(* CODESYS project plc_chalet_vision_fw15.library
   Title: CHALET_Vision
   Version: 3.0.1
   Placeholder: CHALET_Vision
   Company: Beckhoff CH

Project tree, tasks and I/O mapping:
  libraries: CHALET_BaseComponents, * (Beckhoff CH); Tc2_EtherCAT, * (Beckhoff Automation GmbH); Tc2_Standard, * (Beckhoff Automation GmbH); Tc2_System, * (Beckhoff Automation GmbH); Tc2_Utilities, * (Beckhoff Automation GmbH); Tc3_EventLogger, * (Beckhoff Automation GmbH); Tc3_Module, * (Beckhoff Automation GmbH); Tc3_Vision, * (Beckhoff Automation GmbH)
  COMPONENTs/
    CameraTriggerController/
      Base FB/
        function block FB_CameraTriggerController_Base [ST]: FB_init, Feedback, NextPossibleTriggerTime, Operational, Reset, SetParent, State, Trigger
        interface I_CameraTriggerController_Base: Feedback, NextPossibleTriggerTime, Operational, Reset, SetParent, State
        interface I_CameraTriggerController_StatusOnly: Feedback, Operational, State
      EL2258 - 8Ch. digital output timestamp/
        function block FB_EL2258_1Ch_TSO [ST]: Duration_1us, Operational, Reset, State, Trigger, TriggerDelay_1ns, Update
      EL2596 - 1Ch. LED output and camera trigger/
        function block FB_EL2596 [ST]: Duration_1us, Operational, Reset, State, Trigger, TriggerDelay_1ns, Update
        interface I_HwTimestamp_Mode: Duration_1us, Trigger, TriggerDelay_1ns
      EtherCAT Timestamp trigger/
        function block FB_EtherCAT_Trigger [ST]: NextPossibleTriggerTime, Operational, Reset, State, Trigger, TriggerDelay_1ns, Update
        function block FB_EtherCAT_Trigger_old [ST]: Operational, Reset, State, Trigger, TriggerDelay_1ns, Update
        interface I_SwTimestamp_Mode: Trigger, TriggerDelay_1ns
      GigE - Softwaretrigger/
        function block FB_GigeSoftwaretrigger [ST]: Duration_1us, GigeCamera, Reset, Trigger, TriggerDelay_1ns, Update
        interface I_GigeSoftTrigger_Mode: GigeCamera, Trigger, TriggerDelay_1ns
    IlluminationController/
      EL2595 - 1Ch. LED output timestamp/
        function block FB_EL2595 [ST]: Busy, Duration_1us, Operational, Reset, State, Trigger, Update
      SingleOutput/
        function block FB_IlluminationSingleOutput [ST]: Busy, Configure, FB_init, Initialize, Operational, Reset, State, Trigger, Update
        interface I_IlluminationSingleOutput_Mode: Duration_1us, Trigger
      VIx2000/
        DUTs/
          data type E_VIx2000_Status
          data type ST_VIx2000_Channel
          data type ST_VIx2000_InDevice
          data type ST_VIx2000_OutDevice
          data type ST_VIx2000_Pulse
        function block FB_VIx2000 [ST]: Busy, Configure, Duration_1us, Enable, Initialize, Operational, Reset, State, Trigger, Update
        interface I_VIx2000_Mode: Configure, Trigger
      function block FB_IlluminationController_Base [ST]: Busy, NextPossibleTriggerTime, Operational, Reset, SetParent, State, Trigger
      interface I_IlluminationController_Base: Busy, NextPossibleTriggerTime, Operational, Reset, SetParent, State
      interface I_IlluminationController_StatusOnly: Busy, Operational, State
    ImageProvider/
      Base FB/
        function block FB_ImageProvider_Base [ST]: FB_init, Feedback, Initialize, Operational, Reset, SetParent, State, TryGetImage
        interface I_ImageProvider_Base: Feedback, Operational, Reset, SetParent, State, TryGetImage
        interface I_ImageProvider_StatusOnly: Feedback, Operational, State
      Camera/
        data type E_CameraRegisters_Beckhoff
        data type E_DeviceDefaultState
        data type E_TriggerSource
        function block FB_GigE_Beckhoff [ST]: DeviceDefaultState, DeviceModeNamel, DeviceSerialNumber, DeviceVendorName, DeviceVersion, Exposure_1us, IPAddress, MacAddress, TriggerSource, FB_init, GevCameraControl, Initialize, OID, Reset, Softtrigger, State, TryGetImage, Update
        function block FB_GigE_Vision [ST]: Exposure_1us, FB_init, GevCameraControl, Initialize, OID, Reset, Softtrigger, State, TryGetImage, Update
        interface I_GigEVision_Mode: Exposure_1us, Softtrigger
        interface I_GigEVision_Register_Connection: OID
      ImageFromFile/
        function block FB_ImageFromFile [ST]: FileSourceControl, Initialize, LastImageFileName, OID, RequestSpecificImageName, Reset, State, Trigger, TryGetImage, Update
        interface I_ImageFromFile_Mode: RequestSpecificImageName, Trigger
    Mode/
      Combined illumination and camera triggers/
        function block FB_VisionMode_Pulse_combined [ST]: Configure, Initialize, LastTriggerTime, Name, TriggerAtDcTime, TriggerNow
        interface I_VisionMode_Pulse_combined: Configure, LastTriggerTime, NextPossibleTriggerTime, TriggerAtDcTime, TriggerNow
      Separate illumination and camera triggers/
        function block FB_VisionMode_Pulse_separate [ST]: Configure, Initialize, LastTriggerTime_Camera, LastTriggerTime_Illumination, Name, TriggerAtDcTime_Camera, TriggerAtDcTime_Illumination, TriggerNow_Camera, TriggerNow_Illumination
        interface I_VisionMode_Pulse_separate: Configure, LastTriggerTime_Camera, LastTriggerTime_Illumination, NextPossibleTriggerTime, TriggerAtDcTime_Camera, TriggerAtDcTime_Illumination, TriggerNow_Camera, TriggerNow_Illumination
      function block FB_VisionMode_Base [ST]: LinkComponents, Name, NextPossibleTriggerTime
      interface I_VisionMode_Base: LinkComponents, Name
      interface I_VisionMode_StatusOnly: Name
    VisionSystem/
      function block FB_VisionSystem [ST]: ActiveMode, CameraController, IlluminationController1, IlluminationController2, ImageProvider, FB_exit, ActiveModeName, SetMode, Busy, Error, FB_init, Initialize, Initialized, OID, Operational, Reset, TaskCycleTimeNs, TryGetImage, Update
      interface I_VisionSystem: ActiveMode, CameraController, IlluminationController1, IlluminationController2, ImageProvider, SetMode, Busy, Error, Initialized, Operational, Reset, TaskCycleTimeNs, TryGetImage
    VnRegister-Access/
      internal/
        function block FB_VnRegister_Base [ST]: Error, FB_init, Initialize, OID, ReadDone, Update, WriteDone
        interface I_VnRegister_Status: ReadDone, WriteDone
      function block FB_VnRegister_Memory [ST]: FB_init, ReadData, Update, WriteData
      function block FB_VnRegister_REAL [ST]: FB_init, Update, Value
      function block FB_VnRegister_UDINT [ST]: FB_init, Update, Value
      function block FB_VnRegister_ULINT [ST]: FB_init, Update, Value
  FUNCTIONs/
    Casting/
      function ToCameraController [ST]
      function ToGigeSoftTrigger_Mode [ST]
      function ToGigEVision_Mode [ST]
      function ToHwTimestamp_Mode [ST]
      function ToIlluminationSingleOutput_Mode [ST]
      function ToImageFromFile_Mode [ST]
      function ToImageProvider [ST]
      function TolluminationController [ST]
      function ToSwTimestamp_Mode [ST]
      function ToVisionMode_Pulse_combined [ST]
      function ToVisionMode_Pulse_separate [ST]
      function ToVIx2000_Mode [ST]
    Color/
      data type E_Color_ARGB
      function F_ColorEnumToVector4 [ST]
    Sharpness/
      function F_VND_Sharpness_SumModifiedLaplace_ULINT [ST]
  TYPEs/
    data type E_StateTerminal
    data type ST_ImageWithInfo
  00000000-0000-0000-0000-000000000000|LICENSE.md
  LICENSE.md
  global variables VisionParameterlist
*)

// COMPONENTs/IlluminationController/VIx2000/DUTs/E_VIx2000_Status
{attribute 'qualified_only'}
{attribute 'strict'}
{attribute 'to_string'}
TYPE E_VIx2000_Status :
(
	INIT := 0,
	READY,
	TRIGGERING,
	ERROR,
	RESET,
	RESETING
):=INIT;
END_TYPE

// COMPONENTs/IlluminationController/VIx2000/DUTs/ST_VIx2000_Channel
TYPE ST_VIx2000_Channel :
STRUCT
	nBrightness 	 : UINT;
	nDuration_1us 	 : UDINT;
END_STRUCT
END_TYPE

// COMPONENTs/IlluminationController/VIx2000/DUTs/ST_VIx2000_InDevice
TYPE ST_VIx2000_InDevice :
STRUCT
	bReady					: BOOL := FALSE;		// Illumination ready
	bWarning				: BOOL := FALSE;		// Illumination has warning
	bError					: BOOL := FALSE;		// Illumination has error
	bDiag					: BOOL := FALSE;		// ???
	nStatus					: UDINT := 0;			// Illumination state
	nSwitch_on_counter		: UDINT := 0;			// Illumination switching counter
END_STRUCT
END_TYPE

// COMPONENTs/IlluminationController/VIx2000/DUTs/ST_VIx2000_OutDevice
TYPE ST_VIx2000_OutDevice :
STRUCT
	bEnable					: BOOL 	:= FALSE;					// Illumination enable
	bReset					: BOOL	:= FALSE;					// Illumination reset
END_STRUCT
END_TYPE

// COMPONENTs/IlluminationController/VIx2000/DUTs/ST_VIx2000_Pulse
TYPE ST_VIx2000_Pulse :
STRUCT
	nTimestamp 		: T_DCTIME64;
	nFlashDelay 	: UINT;
END_STRUCT
END_TYPE

// COMPONENTs/ImageProvider/Camera/E_CameraRegisters_Beckhoff
{attribute 'qualified_only'}
{attribute 'to_string'}
TYPE E_CameraRegisters_Beckhoff :
(
BootStrap_VersionMajor_BootStrap_VersionMinor := 16#00000000, // GigE Vision Minor Version
BootStrap_DeviceEndianess_BootStrap_CharacterSet := 16#00000004, // BootStrap CharacterSet
BootStrap_MACAddress_High      := 16#00000008, // None
BootStrap_MACAddress_Low       := 16#0000000C, // None
BootStrap_SupportedLLA_BootStrap_SupportedDHCP_BootStrap_SupportedPersistentIP := 16#00000010, // PersistentIP Register
BootStrap_EnabledDHCP_BootStrap_EnabledPersistentIP_BootStrap_EnabledLLA := 16#00000014, // LLA Register Enabled
BootStrap_IPAddress            := 16#00000024, // Current IP Address Register
BootStrap_SubnetMask           := 16#00000034, // Current Subnet Mask Register
BootStrap_Gateway              := 16#00000044, // Current Subnet Mask Register
DeviceVendorName               := 16#00000048, // Name of the camera vendor which is always Beckhoff Automation GmbH & Co.KG
DeviceModelName                := 16#00000068, // Displays the device model name.
DeviceVersion                  := 16#00000088, // Displays the device version which includes the firmware release and build.
DeviceSerialNumber             := 16#000000D8, // Displays the factory set camera serial number.
DeviceUserID                   := 16#000000E8, // A user set ID of up to 15 characters. By default this field is set to the serial number of the camera.
GevFirstURL                    := 16#00000200, // NULL-terminated string providing the first URL to the XML device description file.
GevSecondURL                   := 16#00000400, // NULL-terminated string providing the second URL to the XML device description file.
BootStrap_NumberOfInterfaces   := 16#00000600, // Number Of Interfaces
BootStrap_PersistentIPAddress  := 16#0000064C, // Persistent IP Address Register
BootStrap_PersistentSubnetMask := 16#0000065C, // Persistent Subnet Mask Register
BootStrap_PersistentDefaultGateway := 16#0000066C, // Persistent Default Gateway Register
BootStrap_MessageChannelCount  := 16#00000900, // Number of Message Channel Register
BootStrap_StreamChannelCount   := 16#00000904, // Number of Stream Channel Register
BootStrap_EVENTDATASupported_BootStrap_WRITEMEMSupported_BootStrap_UserDefinedNameSupported_BootStrap_SerialNumberSupported_BootStrap_ConcatenationSupported_BootStrap_PACKETRESENDSupported_BootStrap_EVENTSupported := 16#00000934, // EVENT Supported
BootStrap_GevHeartbeatTimeout  := 16#00000938, // Current heartbeat timeout in milliseconds
BootStrap_TimestampTickFrequencyHigh := 16#0000093C, // 32-MSB of the timestamp Frequency
BootStrap_TimestampTickFrequencyLow := 16#00000940, // 32-LSB of the timestamp Frequencyy
BootStrap_GevTimestampControl  := 16#00000944, // Timestamp Control Register
BootStrap_TimestampValueHigh   := 16#00000948, // 32-MSB of the timestamp Value
BootStrap_TimestampValueLow    := 16#0000094C, // 32-LSB of the timestamp Value
BootStrap_GVSPExtendedID       := 16#00000960, // GVSP Extended ID
pGevSCPSPacketSizeReg          := 16#00000D04, // None
pGevSCPDReg                    := 16#00000D08, // Inter-Packet Delay
pPhysicalWidthReg              := 16#10000008, // None
pPhysicalHeightReg             := 16#1000000C, // None
pSensorPixelWidthReg           := 16#10000010, // None
pSensorPixelHeightReg          := 16#10000014, // None
pDeviceScanTypeReg             := 16#10000018, // None
pSensorShutterModeReg          := 16#1000001C, // None
pMaxThroughputReg              := 16#10000020, // None
pPixelFormatReg                := 16#10000034, // None
pAcquisitionModeReg            := 16#10000040, // None
pAcquisitionFrameCountReg      := 16#10000044, // None
pSensorColorReg                := 16#10000048, // True, if a color sensor has been detected.
pSensorPolarizationReg         := 16#1000004C, // True, if a polarization sensor has been detected.
pAcquisitionStartReg           := 16#100000A8, // None
pAcquisitionStopReg            := 16#100000AC, // None
pAcquisitionAbortReg           := 16#100000B0, // None
SensorName                     := 16#10000150, // Displays the model of the sensor.
pAcquisitionStatusBaseReg      := 16#10000204, // None
pAcquisitionStatusAcquisitionActiveReg := 16#10000208, // None
pRegion0WidthReg               := 16#10000300, // None
pRegion1WidthReg               := 16#10000304, // None
pRegion2WidthReg               := 16#10000308, // None
pRegion3WidthReg               := 16#1000030C, // None
pRegion4WidthReg               := 16#10000310, // None
pRegion5WidthReg               := 16#10000314, // None
pRegion6WidthReg               := 16#10000318, // None
pRegion7WidthReg               := 16#1000031C, // None
pRegion0MinWidthReg            := 16#10000330, // None
pRegion1MinWidthReg            := 16#10000334, // None
pRegion2MinWidthReg            := 16#10000338, // None
pRegion3MinWidthReg            := 16#1000033C, // None
pRegion4MinWidthReg            := 16#10000340, // None
pRegion5MinWidthReg            := 16#10000344, // None
pRegion6MinWidthReg            := 16#10000348, // None
pRegion7MinWidthReg            := 16#1000034C, // None
pRegion0MaxWidthReg            := 16#10000360, // None
pRegion1MaxWidthReg            := 16#10000364, // None
pRegion2MaxWidthReg            := 16#10000368, // None
pRegion3MaxWidthReg            := 16#1000036C, // None
pRegion4MaxWidthReg            := 16#10000370, // None
pRegion5MaxWidthReg            := 16#10000374, // None
pRegion6MaxWidthReg            := 16#10000378, // None
pRegion7MaxWidthReg            := 16#1000037C, // None
pRegion0IncWidthReg            := 16#10000390, // None
pRegion1IncWidthReg            := 16#10000394, // None
pRegion2IncWidthReg            := 16#10000398, // None
pRegion3IncWidthReg            := 16#1000039C, // None
pRegion4IncWidthReg            := 16#10000400, // None
pRegion5IncWidthReg            := 16#10000404, // None
pRegion6IncWidthReg            := 16#10000408, // None
pRegion7IncWidthReg            := 16#1000040C, // None
pRegion0HeightReg              := 16#10000500, // None
pRegion1HeightReg              := 16#10000504, // None
pRegion2HeightReg              := 16#10000508, // None
pRegion3HeightReg              := 16#1000050C, // None
pRegion4HeightReg              := 16#10000510, // None
pRegion5HeightReg              := 16#10000514, // None
pRegion6HeightReg              := 16#10000518, // None
pRegion7HeightReg              := 16#1000051C, // None
pRegion0MinHeightReg           := 16#10000530, // None
pRegion1MinHeightReg           := 16#10000534, // None
pRegion2MinHeightReg           := 16#10000538, // None
pRegion3MinHeightReg           := 16#1000053C, // None
pRegion4MinHeightReg           := 16#10000540, // None
pRegion5MinHeightReg           := 16#10000544, // None
pRegion6MinHeightReg           := 16#10000548, // None
pRegion7MinHeightReg           := 16#1000054C, // None
pRegion0MaxHeightReg           := 16#10000560, // None
pRegion1MaxHeightReg           := 16#10000564, // None
pRegion2MaxHeightReg           := 16#10000568, // None
pRegion3MaxHeightReg           := 16#1000056C, // None
pRegion4MaxHeightReg           := 16#10000570, // None
pRegion5MaxHeightReg           := 16#10000574, // None
pRegion6MaxHeightReg           := 16#10000578, // None
pRegion7MaxHeightReg           := 16#1000057C, // None
pRegion0IncHeightReg           := 16#10000590, // None
pRegion1IncHeightReg           := 16#10000594, // None
pRegion2IncHeightReg           := 16#10000598, // None
pRegion3IncHeightReg           := 16#1000059C, // None
pRegion4IncHeightReg           := 16#10000600, // None
pRegion5IncHeightReg           := 16#10000604, // None
pRegion6IncHeightReg           := 16#10000608, // None
pRegion7IncHeightReg           := 16#1000060C, // None
pRegion0OffsetXReg             := 16#10000800, // None
pRegion1OffsetXReg             := 16#10000804, // None
pRegion2OffsetXReg             := 16#10000808, // None
pRegion3OffsetXReg             := 16#1000080C, // None
pRegion4OffsetXReg             := 16#10000810, // None
pRegion5OffsetXReg             := 16#10000814, // None
pRegion6OffsetXReg             := 16#10000818, // None
pRegion7OffsetXReg             := 16#1000081C, // None
pRegion0MinOffsetXReg          := 16#10000830, // None
pRegion1MinOffsetXReg          := 16#10000834, // None
pRegion2MinOffsetXReg          := 16#10000838, // None
pRegion3MinOffsetXReg          := 16#1000083C, // None
pRegion4MinOffsetXReg          := 16#10000840, // None
pRegion5MinOffsetXReg          := 16#10000844, // None
pRegion6MinOffsetXReg          := 16#10000848, // None
pRegion7MinOffsetXReg          := 16#1000084C, // None
pRegion0MaxOffsetXReg          := 16#10000860, // None
pRegion1MaxOffsetXReg          := 16#10000864, // None
pRegion2MaxOffsetXReg          := 16#10000868, // None
pRegion3MaxOffsetXReg          := 16#1000086C, // None
pRegion4MaxOffsetXReg          := 16#10000870, // None
pRegion5MaxOffsetXReg          := 16#10000874, // None
pRegion6MaxOffsetXReg          := 16#10000878, // None
pRegion7MaxOffsetXReg          := 16#1000087C, // None
pRegion0IncOffsetXReg          := 16#10000890, // None
pRegion1IncOffsetXReg          := 16#10000894, // None
pRegion2IncOffsetXReg          := 16#10000898, // None
pRegion3IncOffsetXReg          := 16#1000089C, // None
pRegion4IncOffsetXReg          := 16#10000900, // None
pRegion5IncOffsetXReg          := 16#10000904, // None
pRegion6IncOffsetXReg          := 16#10000908, // None
pRegion7IncOffsetXReg          := 16#1000090C, // None
pRegion0OffsetYReg             := 16#10000A00, // None
pRegion1OffsetYReg             := 16#10000A04, // None
pRegion2OffsetYReg             := 16#10000A08, // None
pRegion3OffsetYReg             := 16#10000A0C, // None
pRegion4OffsetYReg             := 16#10000A10, // None
pRegion5OffsetYReg             := 16#10000A14, // None
pRegion6OffsetYReg             := 16#10000A18, // None
pRegion7OffsetYReg             := 16#10000A1C, // None
pRegion0MinOffsetYReg          := 16#10000A30, // None
pRegion1MinOffsetYReg          := 16#10000A34, // None
pRegion2MinOffsetYReg          := 16#10000A38, // None
pRegion3MinOffsetYReg          := 16#10000A3C, // None
pRegion4MinOffsetYReg          := 16#10000A40, // None
pRegion5MinOffsetYReg          := 16#10000A44, // None
pRegion6MinOffsetYReg          := 16#10000A48, // None
pRegion7MinOffsetYReg          := 16#10000A4C, // None
pRegion0MaxOffsetYReg          := 16#10000A60, // None
pRegion1MaxOffsetYReg          := 16#10000A64, // None
pRegion2MaxOffsetYReg          := 16#10000A68, // None
pRegion3MaxOffsetYReg          := 16#10000A6C, // None
pRegion4MaxOffsetYReg          := 16#10000A70, // None
pRegion5MaxOffsetYReg          := 16#10000A74, // None
pRegion6MaxOffsetYReg          := 16#10000A78, // None
pRegion7MaxOffsetYReg          := 16#10000A7C, // None
pRegion0IncOffsetYReg          := 16#10000A90, // None
pRegion1IncOffsetYReg          := 16#10000A94, // None
pRegion2IncOffsetYReg          := 16#10000A98, // None
pRegion3IncOffsetYReg          := 16#10000A9C, // None
pRegion4IncOffsetYReg          := 16#10000B00, // None
pRegion5IncOffsetYReg          := 16#10000B04, // None
pRegion6IncOffsetYReg          := 16#10000B08, // None
pRegion7IncOffsetYReg          := 16#10000B0C, // None
DeviceFirmwareVersion          := 16#10010000, // Displays the currently loaded firmware version manufacturer's code.
pSensorHorizontalDriveModeReg  := 16#11000010, // None
pSensorVerticalDriveModeReg    := 16#11000014, // None
pGevSCPDMinReg                 := 16#12000D08, // Minimum Inter-Packet Delay register
pGevSCPDMaxReg                 := 16#12100D08, // Maximum Inter-Packet Delay register
pGevSCPDIncReg                 := 16#12200D08, // Increment Inter-Packet Delay register
pGevIPConfigurationStatusReg   := 16#20000000, // None
pFrameRateReg                  := 16#30000008, // None
pAcquisitionFrameRateEnableReg := 16#30000010, // None
pGainReg                       := 16#30000014, // None
pOffsetReg                     := 16#3000001C, // None
pExposureModeReg               := 16#30000020, // None
pExposureTimeReg               := 16#30000024, // None
ReverseX_Reg                   := 16#3000005C, // None
ReverseY_Reg                   := 16#30000060, // None
pPixelColorFilterReg           := 16#30000064, // None
pBalanceRatioReg               := 16#30000104, // None
pBalanceRatioRedReg            := 16#30000108, // None
pBalanceRatioGreenReg          := 16#3000010C, // None
pBalanceRatioBlueReg           := 16#30000110, // None
pGammaReg                      := 16#30000300, // None
pTestPatternCountReg           := 16#30000404, // None
pTestPatternReg                := 16#30000408, // None
pTestPatternModeReg            := 16#3000040C, // None
pTestPatternParameter1Reg      := 16#30000410, // None
pTestPatternParameter2Reg      := 16#30000414, // None
pTestPatternHorizontalPositionReg := 16#30000418, // None
pTestPatternVerticalPositionReg := 16#3000041C, // None
pTestPatternHorizontalStepSizeReg := 16#30000420, // None
pTestPatternVerticalStepSizeReg := 16#30000424, // None
pTestPatternHorizontalNumReg   := 16#30000428, // None
pTestPatternVerticalNumReg     := 16#3000042C, // None
pTestPatternColorWidthReg      := 16#30000430, // None
pTestPatternBackGroundReg      := 16#30000434, // None
pTestPatternGradientStepReg    := 16#30000438, // None
pTestPatternParameterMaskReg   := 16#30000440, // None
TestPatternDescription         := 16#30001000, // None
UserSetDescription             := 16#30001120, // Description of the selected User Set content.
UserSetDescription1            := 16#30001140, // Description of the selected User Set content.
UserSetDescription2            := 16#30001160, // Description of the selected User Set content.
UserSetDescription3            := 16#30001180, // Description of the selected User Set content.
UserSetDescription4            := 16#300011A0, // Description of the selected User Set content.
pUserSet0LoadReg               := 16#30001200, // None
pUserSet1LoadReg               := 16#30001204, // None
pUserSet2LoadReg               := 16#30001208, // None
pUserSet3LoadReg               := 16#3000120C, // None
pUserSet4LoadReg               := 16#30001210, // None
pUserSet0SaveReg               := 16#30001300, // None
pUserSet1SaveReg               := 16#30001304, // None
pUserSet2SaveReg               := 16#30001308, // None
pUserSet3SaveReg               := 16#3000130C, // None
pUserSet4SaveReg               := 16#30001310, // None
pUserSetDefaultReg             := 16#30001500, // None
pUserSetFeatureEnableReg       := 16#30001510, // None
pRegionsAvailableReg           := 16#30010000, // Maximum regions of interest available.
pSensorROIMinimumHorizontalValueReg := 16#30010100, // The minimum horizontal value register
pSensorROIMinimumVerticalValueReg := 16#30010104, // The minimum vertical value register
pSensorROIMaximumHorizontalValueReg := 16#30010108, // The maximum horizontal value register
pSensorROIMaximumVerticalValueReg := 16#3001010C, // The maximum vertical value register
pRegionModeReg                 := 16#30010800, // Region Mode base register.
pRegion1ModeReg                := 16#30010804, // Region Mode 1 register.
pRegion2ModeReg                := 16#30010808, // Region Mode 2 register.
pRegion3ModeReg                := 16#3001080C, // Region Mode 3 register.
pRegion4ModeReg                := 16#30010810, // Region Mode 4 register.
pRegion5ModeReg                := 16#30010814, // Region Mode 5 register.
pRegion6ModeReg                := 16#30010818, // Region Mode 6 register.
pRegion7ModeReg                := 16#3001081C, // Region Mode 7 register.
pLineModeReg                   := 16#30020040, // None
pLineInverterReg               := 16#30030040, // None
pLineStatus                    := 16#30040040, // None
pTriggerModeBaseReg            := 16#31000100, // None
pSoftwareTriggerAcquisitionStartReg := 16#31000104, // None
pTriggerSourceBaseReg          := 16#31000108, // None
pTriggerActivationAcquisitionStartReg := 16#3100010C, // None
pTriggerDelayAcquisitionStartReg := 16#31000110, // None
pTriggerModeFrameStartReg      := 16#31000400, // None
pSoftwareTriggerFrameStartReg  := 16#31000404, // None
pTriggerSourceFrameStartReg    := 16#31000408, // None
pTriggerActivationFrameStartReg := 16#3100040C, // None
pTriggerDelayFrameStartReg     := 16#31000410, // None
pFrameRateRegMax               := 16#31001020, // None
pExposureTimeMaxReg            := 16#31001024, // None
pFrameRateRegMin               := 16#31001028, // None
pExposureTimeMinReg            := 16#3100102C, // None
pHorizontalBinningReg          := 16#31001030, // None
pVerticalBinningReg            := 16#31001034, // None
pOpticControllerPresentReg     := 16#32000004, // None
pOpticControllerStatusReg      := 16#32000008, // None
pObjectSensorDistanceReg       := 16#32000010, // Object Sensor Distance Register
pDeviceConnectionSpeedReg      := 16#32100010, // None
pDeviceConnectionStatusReg     := 16#32100014, // None
pDeviceResetReg                := 16#32100018, // None
pDeviceIndicatorModeReg        := 16#32110000, // None
pDeviceStateReg                := 16#32110004, // None
pDeviceDefaultStateReg         := 16#32110008, // None
pLightControllerPresentReg     := 16#33000004, // None
pLightConnectionStatusReg      := 16#33000008, // None
pLightController0Channel1TriggerActiveReg := 16#33000110, // Trigger channel 1 active register
pLightController0Channel2TriggerActiveReg := 16#33000114, // Trigger channel 2 active register
pLightController0Channel3TriggerActiveReg := 16#33000118, // Trigger channel 3 active register
pLightController0Channel4TriggerActiveReg := 16#3300011C, // Trigger channel 4 active register
pLightController0Channel1BrightnessReg := 16#33000120, // Brightness register of channel 1
pLightController0Channel2BrightnessReg := 16#33000124, // Brightness register of channel 2
pLightController0Channel3BrightnessReg := 16#33000128, // Brightness register of channel 3
pLightController0Channel4BrightnessReg := 16#3300012C, // Brightness register of channel 4
pLightController0Channel1TriggerModeReg := 16#33000130, // None
pLightController0Channel2TriggerModeReg := 16#33000134, // None
pLightController0Channel3TriggerModeReg := 16#33000138, // None
pLightController0Channel4TriggerModeReg := 16#3300013C, // None
pLightController0Channel1TriggerDurationReg := 16#33000140, // None
pLightController0Channel2TriggerDurationReg := 16#33000144, // None
pLightController0Channel3TriggerDurationReg := 16#33000148, // None
pLightController0Channel4TriggerDurationReg := 16#3300014C, // None
pLightController0Channel1TriggerDelayReg := 16#33000150, // None
pLightController0Channel2TriggerDelayReg := 16#33000154, // None
pLightController0Channel3TriggerDelayReg := 16#33000158, // None
pLightController0Channel4TriggerDelayReg := 16#3300015C, // None
LightController0Channel1Color  := 16#33001000, // The color of the emitted light.
LightController0Channel2Color  := 16#33001014, // The color of the emitted light.
LightController0Channel3Color  := 16#33001028, // The color of the emitted light.
LightController0Channel4Color  := 16#3300103C, // The color of the emitted light.
pLightControllerEnabledReg     := 16#33100000, // None
pLightControllerPowerGoodReg   := 16#33100004, // None
pLUTEnabledReg                 := 16#35000000, // None
pTransferBlockDurationLowReg   := 16#35000100, // None
pTransferBlockDurationHighReg  := 16#35000104, // None
pTLParamsLockedReg             := 16#35000108, // Features locked during acquisition
pPayloadSizeReg                := 16#3500010C, // None
pPacketSizeMinReg              := 16#36000100, // Minimum packet size register
pPacketSizeMaxReg              := 16#36000104, // Maximum packet size register
pPacketSizeIncReg              := 16#36000108, // Increment of packet size register
pCounter0EventSourceReg        := 16#37000100, // Counter0 Event Source Reg
pCounter1EventSourceReg        := 16#37000104, // Counter1 Event Source Reg
pCounter2EventSourceReg        := 16#37000108, // Counter2 Event Source Reg
pCounter3EventSourceReg        := 16#3700010C, // Counter3 Event Source Reg
pCounter4EventSourceReg        := 16#37000110, // Counter4 Event Source Reg
pCounter5EventSourceReg        := 16#37000114, // Counter5 Event Source Reg
pCounter0ResetReg              := 16#37000200, // Counter0 Reset Reg
pCounter1ResetReg              := 16#37000204, // Counter1 Reset Reg
pCounter2ResetReg              := 16#37000208, // Counter2 Reset Reg
pCounter3ResetReg              := 16#3700020C, // Counter3 Reset Reg
pCounter4ResetReg              := 16#37000210, // Counter4 Reset Reg
pCounter5ResetReg              := 16#37000214, // Counter5 Reset Reg
pCounter0ValueReg              := 16#37000300, // Counter0 Value Reg
pCounter1ValueReg              := 16#37000304, // Counter1 Value Reg
pCounter2ValueReg              := 16#37000308, // Counter2 Value Reg
pCounter3ValueReg              := 16#3700030C, // Counter3 Value Reg
pCounter4ValueReg              := 16#37000310, // Counter4 Value Reg
pCounter5ValueReg              := 16#37000314, // Counter5 Value Reg
pDeviceTemperatureBaseReg      := 16#40000004, // None
pDeviceTemperatureCoreReg      := 16#40000008, // None
pDeviceTemperaturePhyReg       := 16#4000000C, // None
pDeviceTemperatureLiquidLensReg := 16#40000010, // None
pTimestampImage                := 16#41000004, // None
pExtendedInternalTimestampControlRegister := 16#41000050, // None
pExtendedEtherCATTimestampControlRegister := 16#41000054, // None
pTimestampRegHigh              := 16#41000100, // None
pDistributedClocksTimestampRegHigh := 16#41000104, // None
pTimestampLatchRegHigh         := 16#41000110, // None
pDistributedClocksTimestampLatchRegHigh := 16#41000114, // None
pTimestampRegLow               := 16#41000200, // None
pDistributedClocksTimestampRegLow := 16#41000204, // None
pTimestampLatchRegLow          := 16#41000210, // None
pDistributedClocksTimestampLatchRegLow := 16#41000214, // None
pEtherCATLinkActiveReg         := 16#50000000, // None
pGevMACAddressHighWordReg := 16#04F91B00, // None
pGevMACAddressLowWordReg := 16#04F91B04 // None
) UDINT;
END_TYPE

// COMPONENTs/ImageProvider/Camera/E_DeviceDefaultState
{attribute 'qualified_only'}
{attribute 'to_string'}
TYPE E_DeviceDefaultState :
(
	AutoDetect		 	:= 0,
	GigE_Vision	 		:= 1,
	EtherCAT_IO			:= 2,
	EtherCAT_Full		:= 3
)UDINT := AutoDetect;
END_TYPE

// COMPONENTs/ImageProvider/Camera/E_TriggerSource
{attribute 'qualified_only'}
{attribute 'to_string'}
TYPE E_TriggerSource :
(
	SoftwareTrigger 	:= 0,
	HardwareInput	 	:= 1,
	EtherCAT			:= 2
)UDINT := SoftwareTrigger;
END_TYPE

// FUNCTIONs/Color/E_Color_ARGB
TYPE E_Color_ARGB : CHALET_BaseComponents.E_Colors_ARGB; END_TYPE

// TYPEs/E_StateTerminal
{attribute 'qualified_only'}
{attribute 'strict'}
{attribute 'to_string'}
TYPE E_StateTerminal :
(
	RESET := 0,
	RESETING,
	INIT := 10,
	READY := 20,
	TRIGGERING := 30,
	ERROR := 100
):=INIT;
END_TYPE

// TYPEs/ST_ImageWithInfo
TYPE ST_ImageWithInfo :
STRUCT
	ipImage			: ITcVnImage;			// Image
	stInfo 			: TcVnImageInfo;		// Image information   
	sCurrentImageFileName : STRING(500);		// Image name.  For a file the file name, for a camera a fictitious name  
	stGvspInfo 		: GVSP_IMAGE_INFO;		// Returns the GVSP (GigE Vision Streaming Protocol) meta information.
END_STRUCT
END_TYPE

// VisionParameterlist
{attribute 'qualified_only'}
VAR_GLOBAL CONSTANT
	(*Maximum GigE-Register read at same time*)
	MAX_VN_REGISTER_READ 			: UDINT := 1;
	
	(*Maximum GigE-Register write at same time*)
	MAX_VN_REGISTER_WRITE 			: UDINT := 1;
	
	(* The state machine for the illuminaton waits in the “Triggering” state until the component has increased the nSwitch_on_counter *)
	ILLUMINATION_WAIT_FOR_TRIGGER_FEEDBACK : BOOL := FALSE;
END_VAR

// COMPONENTs/CameraTriggerController/Base FB/FB_CameraTriggerController_Base
{attribute 'no_explicit_call' := 'Do not call the body - Stick to OOP'}
FUNCTION_BLOCK ABSTRACT FB_CameraTriggerController_Base EXTENDS FB_CH_Object IMPLEMENTS I_CameraTriggerController_Base
VAR
	ipVisionSystem		: I_VisionSystem;			//Interface to "Owner" of this module. Visionsystem
	fbAlarmGeneral 		: FB_TcAlarm;				// Terminal general alarm
	{attribute 'hide'}  						
	fbFeedback 				: FB_CH_Feedback(THIS^.fbSourceInfo);
END_VAR

METHOD FB_init : BOOL
VAR_INPUT
	bInitRetains : BOOL; // if TRUE, the retain variables are initialized (warm start / cold start)
	bInCopyCode : BOOL;  // if TRUE, the instance afterwards gets moved into the copy code (online change)
END_VAR
VAR_INST
	{attribute 'hide'}
	bFBInitCalledOnce : BOOL; //Do the following code once during start up and not during onlinechange
END_VAR
//Do the following code once during start up and not during onlinechange
IF NOT bFBInitCalledOnce THEN 
	
	;

END_IF

bFBInitCalledOnce := TRUE;
END_METHOD

{attribute 'monitoring':='call'}
PROPERTY Feedback : I_CH_Feedback
GET
Feedback := THIS^.fbFeedback;
END_GET
END_PROPERTY

{attribute 'monitoring' := 'call'}
PROPERTY NextPossibleTriggerTime : T_DCTIME64
GET
VAR
	nEtherCatCycles 	: UINT;	
END_VAR
//If attribute 'TcCallAfterOutputUpdate' is set, it takes 1 cycle more to send timestamp to hardware
IF TwinCAT_SystemInfoVarList._TaskInfo[THIS^.TaskIndex].InCallAfterOutputUpdate THEN
	nEtherCatCycles := 3;
ELSE
	nEtherCatCycles := 2;
END_IF


NextPossibleTriggerTime := F_GetCurDcTaskTime64()(*1ns*) + (THIS^.ipVisionSystem.TaskCycleTimeNs(*1ns*) * nEtherCatCycles (*Cycles*)) + 300_000(*300us(determined by testing)*);
END_GET
END_PROPERTY

{attribute 'monitoring' := 'call'}
PROPERTY Operational : BOOL
GET
Operational := TRUE;
END_GET
END_PROPERTY

METHOD ABSTRACT Reset : HRESULT
END_METHOD

METHOD SetParent
VAR_INPUT
	ipVisionSystem  : I_VisionSystem;
END_VAR
THIS^.ipVisionSystem := ipVisionSystem;
END_METHOD

{attribute 'monitoring' := 'call'}
PROPERTY PUBLIC State : E_StateTerminal
GET
State := E_StateTerminal.READY;
END_GET
END_PROPERTY

METHOD ABSTRACT Trigger : HRESULT
VAR_INPUT
	//The data type T_DCTIME64 represents the distributed clock system time (abbreviated as DC time) as a linear 64-bit integer value. 
	//The time is expressed in nanoseconds since 1/1/2000 UTC. The smallest unit is a nanosecond.
	//F_GetCurDcTickTime64()
	nDCTimeStamp	: T_DCTIME64;
END_VAR
END_METHOD

END_FUNCTION_BLOCK

// COMPONENTs/CameraTriggerController/Base FB/I_CameraTriggerController_Base
INTERFACE I_CameraTriggerController_Base EXTENDS I_CH_Object, I_CameraTriggerController_StatusOnly, __SYSTEM.IQueryInterface

{attribute 'monitoring':='call'}
PROPERTY Feedback : I_CH_Feedback
GET
END_GET
END_PROPERTY

{attribute 'monitoring' := 'call'}
PROPERTY NextPossibleTriggerTime : T_DCTIME64
GET
END_GET
END_PROPERTY

{attribute 'monitoring' := 'call'}
PROPERTY Operational : BOOL
GET
END_GET
END_PROPERTY

METHOD Reset : HRESULT
END_METHOD

METHOD SetParent
VAR_INPUT
	ipVisionSystem  : I_VisionSystem;
END_VAR
END_METHOD

{attribute 'monitoring' := 'call'}
PROPERTY PUBLIC State : E_StateTerminal
GET
END_GET
END_PROPERTY

END_INTERFACE

// COMPONENTs/CameraTriggerController/Base FB/I_CameraTriggerController_StatusOnly
INTERFACE I_CameraTriggerController_StatusOnly EXTENDS __SYSTEM.IQueryInterface

{attribute 'monitoring':='call'}
PROPERTY Feedback : I_CH_Feedback
GET
END_GET
END_PROPERTY

{attribute 'monitoring' := 'call'}
PROPERTY Operational : BOOL
GET
END_GET
END_PROPERTY

{attribute 'monitoring' := 'call'}
PROPERTY PUBLIC State : E_StateTerminal
GET
END_GET
END_PROPERTY

END_INTERFACE

// COMPONENTs/VisionSystem/I_VisionSystem
INTERFACE I_VisionSystem EXTENDS I_CH_Object

{attribute 'monitoring' := 'call'}
PROPERTY ActiveMode : I_VisionMode_StatusOnly
GET
END_GET
END_PROPERTY

{attribute 'monitoring' := 'call'}
PROPERTY CameraController : I_CameraTriggerController_StatusOnly
GET
END_GET
END_PROPERTY

{attribute 'monitoring' := 'call'}
PROPERTY IlluminationController1 : I_IlluminationController_StatusOnly
GET
END_GET
END_PROPERTY

{attribute 'monitoring' := 'call'}
PROPERTY IlluminationController2 : I_IlluminationController_StatusOnly
GET
END_GET
END_PROPERTY

{attribute 'monitoring' := 'call'}
PROPERTY ImageProvider : I_ImageProvider_StatusOnly
GET
END_GET
END_PROPERTY

METHOD SetMode : HRESULT
VAR_INPUT
	ipAnyMode : I_VisionMode_Base;
END_VAR
END_METHOD

{attribute 'monitoring' := 'call'}
//Module already has a task - already a trigger active
PROPERTY ABSTRACT Busy : BOOL
GET
END_GET
END_PROPERTY

{attribute 'monitoring' := 'call'}
PROPERTY Error : BOOL  // Module started successfully and entered aquiring mode
GET
END_GET
END_PROPERTY

{attribute 'monitoring':='call'}
PROPERTY Initialized : BOOL
GET
END_GET
END_PROPERTY

{attribute 'monitoring' := 'call'}
PROPERTY PUBLIC Operational : BOOL // Module started successfully and entered aquiring mode
GET
END_GET
END_PROPERTY

METHOD Reset : HRESULT
VAR_INPUT
END_VAR
END_METHOD

{attribute 'monitoring' := 'call'}
PROPERTY TaskCycleTimeNs : UDINT // Set task cycle time in multiples of 100 ns
GET
END_GET
END_PROPERTY

METHOD TryGetImage : HRESULT
VAR_INPUT
	stImageWithInfo : REFERENCE TO ST_ImageWithInfo;
END_VAR
END_METHOD

END_INTERFACE

// COMPONENTs/Mode/I_VisionMode_StatusOnly
INTERFACE I_VisionMode_StatusOnly EXTENDS __SYSTEM.IQueryInterface

{attribute 'monitoring' := 'call'}
// Name or description of this mode
PROPERTY Name : STRING
GET
END_GET
END_PROPERTY

END_INTERFACE

// COMPONENTs/IlluminationController/I_IlluminationController_StatusOnly
INTERFACE I_IlluminationController_StatusOnly EXTENDS  __SYSTEM.IQueryInterface

{attribute 'monitoring' := 'call'}
PROPERTY Busy : BOOL
GET
END_GET
END_PROPERTY

{attribute 'monitoring' := 'call'}
PROPERTY Operational : BOOL
GET
END_GET
END_PROPERTY

{attribute 'monitoring' := 'call'}
PROPERTY PUBLIC State : E_StateTerminal
GET
END_GET
END_PROPERTY

END_INTERFACE

// COMPONENTs/ImageProvider/Base FB/I_ImageProvider_StatusOnly
INTERFACE I_ImageProvider_StatusOnly EXTENDS __SYSTEM.IQueryInterface

{attribute 'monitoring':='call'}
PROPERTY Feedback : I_CH_Feedback
GET
END_GET
END_PROPERTY

{attribute 'monitoring' := 'call'}
PROPERTY PUBLIC Operational : BOOL
// Module started successfully and entered aquiring mode
GET
END_GET
END_PROPERTY

{attribute 'monitoring' := 'call'}
PROPERTY State : ETcVnCameraState
GET
END_GET
END_PROPERTY

END_INTERFACE

// COMPONENTs/Mode/I_VisionMode_Base
INTERFACE I_VisionMode_Base EXTENDS I_CH_Object, I_VisionMode_StatusOnly, __SYSTEM.IQueryInterface

METHOD LinkComponents : HRESULT
VAR_INPUT
	ipVisionSystem				: I_VisionSystem;
	ipCameraTriggerController	: I_CameraTriggerController_Base;
	ipImageProvider 			: I_ImageProvider_Base;	
	ipIlluminationController1 : I_IlluminationController_Base;
	ipIlluminationController2 : I_IlluminationController_Base;
END_VAR
END_METHOD

{attribute 'monitoring' := 'call'}
// Name or description of this mode
PROPERTY Name : STRING
GET
END_GET
END_PROPERTY

END_INTERFACE

// COMPONENTs/ImageProvider/Base FB/I_ImageProvider_Base
INTERFACE I_ImageProvider_Base EXTENDS I_CH_Object, I_ImageProvider_StatusOnly, __SYSTEM.IQueryInterface

{attribute 'monitoring':='call'}
PROPERTY Feedback : I_CH_Feedback
GET
END_GET
END_PROPERTY

{attribute 'monitoring' := 'call'}
PROPERTY PUBLIC Operational : BOOL
// Module started successfully and entered aquiring mode
GET
END_GET
END_PROPERTY

METHOD Reset : HRESULT
END_METHOD

METHOD SetParent
VAR_INPUT
	ipObject : I_CH_Object;
END_VAR
END_METHOD

{attribute 'monitoring' := 'call'}
PROPERTY State : ETcVnCameraState
GET
END_GET
END_PROPERTY

METHOD TryGetImage : HRESULT
VAR_INPUT
	stImageWithInfo	: REFERENCE TO ST_ImageWithInfo;
END_VAR
END_METHOD

END_INTERFACE

// COMPONENTs/IlluminationController/I_IlluminationController_Base
INTERFACE I_IlluminationController_Base EXTENDS I_CH_Object, I_IlluminationController_StatusOnly, __SYSTEM.IQueryInterface

{attribute 'monitoring' := 'call'}
PROPERTY Busy : BOOL
GET
END_GET
END_PROPERTY

{attribute 'monitoring' := 'call'}
PROPERTY NextPossibleTriggerTime : T_DCTIME64
GET
END_GET
END_PROPERTY

{attribute 'monitoring' := 'call'}
PROPERTY Operational : BOOL
GET
END_GET
END_PROPERTY

METHOD Reset : HRESULT
END_METHOD

METHOD SetParent
VAR_INPUT
	ipVisionSystem  : I_VisionSystem;
END_VAR
END_METHOD

{attribute 'monitoring' := 'call'}
PROPERTY PUBLIC State : E_StateTerminal
GET
END_GET
END_PROPERTY

END_INTERFACE

// COMPONENTs/CameraTriggerController/EL2258 - 8Ch. digital output timestamp/FB_EL2258_1Ch_TSO
{attribute 'no_explicit_call' := 'Do not call the body - Stick to OOP'}
FUNCTION_BLOCK FB_EL2258_1Ch_TSO EXTENDS FB_CameraTriggerController_Base IMPLEMENTS I_HwTimestamp_Mode
VAR
	bOutput					AT %Q* 	: BOOL;					// Desired State of Output
	nStartTime 				AT %Q*	: T_DCTIME64;			// Trigger time stamp
	nActivate				AT %Q*	: USINT; 				// 0 -> 3 use new time in terminal
	
	nImpulseLength 			: UDINT := 20000;   	// Impulse length of the lighting period [in 1us]	
	nTriggerDelay 			: UDINT := 0;			// The given trigger time is delayed by this value. E.g. to wait for the maximum lighting value before taking a picture  [in 1ns]
	{attribute 'hide'}
	eState					: E_StateTerminal;				// Current terminal state
	eTriggerSubState		:(SEQ_WirteTime, SEQ_Activate, SEQ_WaitForTriggerDone, SEQ_TriggerOff, SEQ_Deactivate, SEQ_Done); //setting the trigger takes several Ethercat cycles
END_VAR

{attribute 'monitoring' := 'call'}
PROPERTY Duration_1us : UDINT
GET
Duration_1us := THIS^.nImpulseLength;
END_GET
SET
THIS^.nImpulseLength := Duration_1us;
END_SET
END_PROPERTY

{attribute 'monitoring' := 'call'}
PROPERTY Operational : BOOL
GET
Operational := (THIS^.eState = E_StateTerminal.READY) OR (THIS^.eState = E_StateTerminal.TRIGGERING);
END_GET
END_PROPERTY

METHOD PUBLIC Reset : HRESULT
VAR_INPUT
END_VAR
IF THIS^.eState = E_StateTerminal.ERROR THEN
	fbFeedback.ActiveCommand := 'Reset';
	fbFeedback.Busy := TRUE;	
	
	THIS^.eState := E_StateTerminal.RESET;
END_IF
END_METHOD

{attribute 'monitoring' := 'call'}
PROPERTY PUBLIC State : E_StateTerminal
GET
State := THIS^.eState;
END_GET
END_PROPERTY

METHOD PUBLIC Trigger : HRESULT
VAR_INPUT
	//The data type T_DCTIME64 represents the distributed clock system time (abbreviated as DC time) as a linear 64-bit integer value. 
	//The time is expressed in nanoseconds since 1/1/2000 UTC. The smallest unit is a nanosecond.
	//F_GetCurDcTickTime64()
	nDCTimeStamp	: T_DCTIME64;
END_VAR
(* Check if the trigger is minimum 3 EtherCat cycles in future *)
IF nDCTimeStamp < THIS^.NextPossibleTriggerTime  THEN
	Trigger := E_FAIL;
	RETURN;
END_IF

(* Check if not in wrong state *)
IF NOT (THIS^.eState = E_StateTerminal.READY) THEN
	Trigger := E_FAIL;
	RETURN;
END_IF

fbFeedback.ActiveCommand := 'Trigger';
fbFeedback.Busy := TRUE;	


THIS^.nStartTime := nDCTimeStamp + THIS^.nTriggerDelay;
THIS^.bOutput := TRUE;
THIS^.nActivate := 0;

THIS^.eTriggerSubState := SEQ_WirteTime;
THIS^.eState := E_StateTerminal.TRIGGERING;
Trigger := S_OK;
END_METHOD

{attribute 'monitoring' := 'call'}
// The given trigger time is delayed by this value. E.g. to wait for the maximum lighting value before taking a picture  [in 1ns]
PROPERTY TriggerDelay_1ns : UDINT
GET
TriggerDelay_1ns := THIS^.nTriggerDelay;
END_GET
SET
THIS^.nTriggerDelay := TriggerDelay_1ns;
END_SET
END_PROPERTY

METHOD PUBLIC Update : HRESULT
VAR_INST
	fbTimeout : TON;
END_VAR
(* Check for terminal errors *)
//IF THIS^.bError AND NOT (THIS^.eState = E_StateTerminal.RESET) THEN 
//	THIS^.eState := E_StateTerminal.ERROR;
//END_IF

(* Handle terminal state machine *)
CASE THIS^.eState OF
	(* Reset all control variables *)
	E_StateTerminal.RESET:
		THIS^.eState := E_StateTerminal.RESETING;
		
	(* Reset all control variables *)
	E_StateTerminal.RESETING:
		THIS^.eState := E_StateTerminal.INIT;	
		
	(* Enable terminal if ready *)
	E_StateTerminal.INIT:			
		THIS^.eState := E_StateTerminal.READY;

	
	(* Terminal is ready *)
	E_StateTerminal.READY:
		fbFeedback.Done := TRUE;	
		
		THIS^.nStartTime := 0;
		THIS^.bOutput := FALSE;
		THIS^.nActivate := 0;
		
	(* Terminal is triggering *)
	E_StateTerminal.TRIGGERING:
		CASE eTriggerSubState OF
			SEQ_WirteTime:
				//Wirte TimeStamp, Output and Activate=0 in .Trigger()
				//The next commands are allowed only in the next Ethercat cycle
				eTriggerSubState := SEQ_Activate;
				
			SEQ_Activate:
				// Activate new time
				THIS^.nActivate := 3;
				eTriggerSubState := SEQ_WaitForTriggerDone;
				
			SEQ_WaitForTriggerDone:
				// Trigger is done and PulsOffTime is done
				IF (F_GetCurDcTaskTime64() >= (THIS^.nStartTime + (THIS^.nImpulseLength*1000)(*1ns*))) THEN
					THIS^.bOutput := FALSE;
					THIS^.nActivate := 0;
					eTriggerSubState := SEQ_TriggerOff;
				END_IF
				
			SEQ_TriggerOff:	
				THIS^.nActivate := 3;
				eTriggerSubState := SEQ_Deactivate;
				
			SEQ_Deactivate:	
				IF (F_GetCurDcTaskTime64()(*1ns*) > THIS^.nStartTime) THEN
					eTriggerSubState := SEQ_Done;
					//Ready for next Trigger
					THIS^.eState := E_StateTerminal.READY;
				END_IF

				
			SEQ_Done:
			;
		END_CASE
	
	
	(* Error occured *)	
	E_StateTerminal.ERROR:
		fbFeedback.HR := E_FAIL;	
		IF NOT THIS^.fbAlarmGeneral.bRaised THEN
			THIS^.fbAlarmGeneral.Raise(0);	
		END_IF
		
		IF (THIS^.fbAlarmGeneral.eConfirmationState = TcEventConfirmationState.Confirmed) THEN
			THIS^.Reset();			
		END_IF			
END_CASE

(* Timeout if an state is to long active *)
fbTimeout.IN := (THIS^.eState = E_StateTerminal.INIT) OR (THIS^.eState = E_StateTerminal.RESETING) OR (THIS^.eState = E_StateTerminal.TRIGGERING);
fbTimeout.PT := T#5S;
fbTimeout();
IF fbTimeout.Q THEN
	THIS^.eState := E_StateTerminal.ERROR;
END_IF
END_METHOD

END_FUNCTION_BLOCK

// COMPONENTs/CameraTriggerController/EL2596 - 1Ch. LED output and camera trigger/I_HwTimestamp_Mode
INTERFACE I_HwTimestamp_Mode EXTENDS __SYSTEM.IQueryInterface

{attribute 'monitoring' := 'call'}
PROPERTY Duration_1us : UDINT
GET
END_GET
SET
END_SET
END_PROPERTY

METHOD PUBLIC Trigger : HRESULT
VAR_INPUT
	//The data type T_DCTIME64 represents the distributed clock system time (abbreviated as DC time) as a linear 64-bit integer value. 
	//The time is expressed in nanoseconds since 1/1/2000 UTC. The smallest unit is a nanosecond.
	//F_GetCurDcTickTime64()
	nDCTimeStamp	: T_DCTIME64;
END_VAR
END_METHOD

{attribute 'monitoring' := 'call'}
// The given trigger time is delayed by this value. E.g. to wait for the maximum lighting value before taking a picture  [in 1ns]
PROPERTY TriggerDelay_1ns : UDINT
GET
END_GET
SET
END_SET
END_PROPERTY

END_INTERFACE

// COMPONENTs/CameraTriggerController/EL2596 - 1Ch. LED output and camera trigger/FB_EL2596
{attribute 'no_explicit_call' := 'Do not call the body - Stick to OOP'}
FUNCTION_BLOCK FB_EL2596 EXTENDS FB_CameraTriggerController_Base IMPLEMENTS I_HwTimestamp_Mode
VAR
	bEnable					AT %Q* 	: BOOL;					// Terminal enable
	bTriggerImage 			AT %Q* 	: BOOL;					// Trigger for lighting and camera	 
	bReset					AT %Q*	: BOOL;					// Terminal reset
	
	TimeStamp 				AT %Q*	: T_DCTIME64;				// Trigger time stamp
	
	bReadyToActivate		AT %I*	: BOOL := FALSE;		// Terminal ready
	bWarning				AT %I*	: BOOL := FALSE;		// Terminal has warning
	bError					AT %I*	: BOOL := FALSE;		// Terminal has error
	nOperationCounter		AT %I*  : USINT := 0;			// Terminal switching counter
	
		 
	bEnableCameraTrigger 	AT %Q* 	: BOOL := TRUE;			// Enable trigger to be used for the camera
	nImpulseLength 			AT %Q* 	: UDINT := 20000;   	// Impulse length of the lighting period [in 1us]
	nTriggerDelay 			AT %Q* 	: UDINT := 10;			// Delay between lighting and camera trigger [in 100ns]

	{attribute 'hide'}
	eState							: E_StateTerminal;		// Current terminal state
	
	{attribute 'hide'}
	nOperationCounterAtTriggerStart			: USINT;				// Old operation counter as reference

END_VAR

{attribute 'monitoring' := 'call'}
PROPERTY Duration_1us : UDINT
GET
Duration_1us := THIS^.nImpulseLength;
END_GET
SET
THIS^.nImpulseLength := Duration_1us;
END_SET
END_PROPERTY

{attribute 'monitoring' := 'call'}
PROPERTY Operational : BOOL
GET
Operational := (THIS^.eState = E_StateTerminal.READY) OR (THIS^.eState = E_StateTerminal.TRIGGERING);
END_GET
END_PROPERTY

METHOD PUBLIC Reset : HRESULT
VAR_INPUT
END_VAR
IF THIS^.bError OR (THIS^.eState = E_StateTerminal.ERROR) THEN
	fbFeedback.ActiveCommand := 'Reset';
	fbFeedback.Busy := TRUE;	
	
	THIS^.eState := E_StateTerminal.RESET;
END_IF
END_METHOD

{attribute 'monitoring' := 'call'}
PROPERTY PUBLIC State : E_StateTerminal
GET
State := THIS^.eState;
END_GET
END_PROPERTY

METHOD PUBLIC Trigger : HRESULT
VAR_INPUT
	//The data type T_DCTIME64 represents the distributed clock system time (abbreviated as DC time) as a linear 64-bit integer value. 
	//The time is expressed in nanoseconds since 1/1/2000 UTC. The smallest unit is a nanosecond.
	//F_GetCurDcTickTime64()
	nDCTimeStamp	: T_DCTIME64;
END_VAR
(* Check if the trigger is minimum 3 EtherCat cycles in future *)
IF nDCTimeStamp < THIS^.NextPossibleTriggerTime  THEN
	Trigger := E_FAIL;
	RETURN;
END_IF

(* Check if not in wrong state *)
IF NOT (THIS^.eState = E_StateTerminal.READY) THEN
	Trigger := E_FAIL;
	RETURN;
END_IF

fbFeedback.ActiveCommand := 'Trigger';
fbFeedback.Busy := TRUE;	


THIS^.nOperationCounterAtTriggerStart := THIS^.nOperationCounter;
THIS^.TimeStamp := nDCTimeStamp;
THIS^.eState := E_StateTerminal.TRIGGERING;
Trigger := S_OK;
END_METHOD

{attribute 'monitoring' := 'call'}
// The given trigger time is delayed by this value. E.g. to wait for the maximum lighting value before taking a picture  [in 1ns]
PROPERTY TriggerDelay_1ns : UDINT
GET
TriggerDelay_1ns := THIS^.nTriggerDelay*100;
END_GET
SET
THIS^.nTriggerDelay := TriggerDelay_1ns/100;
END_SET
END_PROPERTY

METHOD PUBLIC Update : HRESULT
VAR_INST
	fbTimeOut : TON;
END_VAR
(* Check for terminal errors *)
IF THIS^.bError AND NOT (THIS^.eState = E_StateTerminal.RESET) THEN 
	THIS^.eState := E_StateTerminal.ERROR;
END_IF

(* Handle terminal state machine *)
CASE THIS^.eState OF
	(* Reset all control variables *)
	E_StateTerminal.RESET:
		THIS^.bReset := TRUE;
		THIS^.bEnable := FALSE;
		THIS^.bTriggerImage := FALSE;
		THIS^.eState := E_StateTerminal.RESETING;
		
	(* Reset all control variables *)
	E_StateTerminal.RESETING:
		THIS^.bReset := FALSE;
		THIS^.bEnable := FALSE;
		THIS^.bTriggerImage := FALSE;
		THIS^.eState := E_StateTerminal.INIT;	
		
	(* Enable terminal if ready *)
	E_StateTerminal.INIT:			
		IF THIS^.bReadyToActivate THEN
			THIS^.bReset := FALSE;
			THIS^.bEnable := TRUE;
			THIS^.fbAlarmGeneral.Clear(0, TRUE);
			THIS^.eState := E_StateTerminal.READY;
		END_IF
	
	(* Terminal is ready *)
	E_StateTerminal.READY:
		fbFeedback.Done := TRUE;	
		
	(* Terminal is triggering *)
	E_StateTerminal.TRIGGERING:
		THIS^.bTriggerImage := TRUE;
		IF THIS^.nOperationCounterAtTriggerStart <> THIS^.nOperationCounter THEN
			THIS^.bTriggerImage := FALSE;
			THIS^.eState := E_StateTerminal.READY;
		END_IF
	
	(* Error occured *)	
	E_StateTerminal.ERROR:
		fbFeedback.HR := E_FAIL;
		IF NOT THIS^.fbAlarmGeneral.bRaised THEN
			THIS^.fbAlarmGeneral.Raise(0);	
		END_IF
		
		IF (THIS^.fbAlarmGeneral.eConfirmationState = TcEventConfirmationState.Confirmed) THEN
			THIS^.Reset();			
		END_IF			
END_CASE

(* Timeout if an state is to long active *)
fbTimeOut.IN := (THIS^.eState = E_StateTerminal.INIT) OR (THIS^.eState = E_StateTerminal.RESETING) OR (THIS^.eState = E_StateTerminal.TRIGGERING);
fbTimeOut.PT := T#5S;
fbTimeOut();
IF fbTimeOut.Q THEN
	THIS^.eState := E_StateTerminal.ERROR;
END_IF
END_METHOD

END_FUNCTION_BLOCK

// COMPONENTs/CameraTriggerController/EtherCAT Timestamp trigger/FB_EtherCAT_Trigger
{attribute 'no_explicit_call' := 'Do not call the body - Stick to OOP'}
FUNCTION_BLOCK FB_EtherCAT_Trigger EXTENDS FB_CameraTriggerController_Base IMPLEMENTS I_SwTimestamp_Mode
VAR
	nStartTime 				AT %Q*	: T_DCTIME64;			// Trigger time stamp
	
	{attribute 'hide'}
	nTriggerDelay 			: UDINT := 0;					// The given trigger time is delayed by this value. E.g. to wait for the maximum lighting value before taking a picture  [in 100ns]
	
	{attribute 'hide'}
	eState					: E_StateTerminal;				// Current terminal state
END_VAR

{attribute 'monitoring' := 'call'}
PROPERTY NextPossibleTriggerTime : T_DCTIME64
GET
VAR
	nEtherCatCycles 	: UINT;	
END_VAR
//If attribute 'TcCallAfterOutputUpdate' is set, it takes 1 cycle more to send timestamp to hardware
IF TwinCAT_SystemInfoVarList._TaskInfo[THIS^.TaskIndex].InCallAfterOutputUpdate THEN
	nEtherCatCycles := 3;
ELSE
	nEtherCatCycles := 2;
END_IF


NextPossibleTriggerTime := F_GetCurDcTaskTime64()(*1ns*) + 3_000_000(*zzz 3ms Beta Firmware*) + (THIS^.ipVisionSystem.TaskCycleTimeNs(*1ns*) * nEtherCatCycles (*Cycles*));
END_GET
END_PROPERTY

{attribute 'monitoring' := 'call'}
PROPERTY Operational : BOOL
GET
Operational := (THIS^.eState = E_StateTerminal.READY) OR (THIS^.eState = E_StateTerminal.TRIGGERING);
END_GET
END_PROPERTY

METHOD PUBLIC Reset : HRESULT
VAR_INPUT
END_VAR
IF THIS^.eState = E_StateTerminal.ERROR THEN
	fbFeedback.ActiveCommand := 'Reset';
	fbFeedback.Busy := TRUE;	

	THIS^.eState := E_StateTerminal.RESET;
END_IF
END_METHOD

{attribute 'monitoring' := 'call'}
PROPERTY PUBLIC State : E_StateTerminal
GET
State := THIS^.eState;
END_GET
END_PROPERTY

METHOD PUBLIC Trigger : HRESULT
VAR_INPUT
	//The data type T_DCTIME64 represents the distributed clock system time (abbreviated as DC time) as a linear 64-bit integer value. 
	//The time is expressed in nanoseconds since 1/1/2000 UTC. The smallest unit is a nanosecond.
	//F_GetCurDcTickTime64()
	nDCTimeStamp	: T_DCTIME64;
END_VAR
(* Check if the trigger is minimum 3 EtherCat cycles in future *)
IF (nDCTimeStamp + THIS^.nTriggerDelay) < THIS^.NextPossibleTriggerTime THEN
	Trigger := E_FAIL;
	RETURN;
END_IF

(* Check if not in wrong state *)
IF NOT (THIS^.eState = E_StateTerminal.READY) THEN
	Trigger := E_FAIL;
	RETURN;
END_IF

fbFeedback.ActiveCommand := 'Trigger';
fbFeedback.Busy := TRUE;	


THIS^.nStartTime := nDCTimeStamp + THIS^.nTriggerDelay;


THIS^.eState := E_StateTerminal.TRIGGERING;
Trigger := S_OK;
END_METHOD

{attribute 'monitoring' := 'call'}
// The given trigger time is delayed by this value. E.g. to wait for the maximum lighting value before taking a picture  [in 1ns]
PROPERTY TriggerDelay_1ns : UDINT
GET
TriggerDelay_1ns := THIS^.nTriggerDelay;
END_GET
SET
THIS^.nTriggerDelay := TriggerDelay_1ns;
END_SET
END_PROPERTY

METHOD PUBLIC Update : HRESULT
VAR_INST
	{attribute 'hide'}
	fbTimeout : TON;
END_VAR
(* Handle terminal state machine *)
CASE THIS^.eState OF
	(* Reset all control variables *)
	E_StateTerminal.RESET:
		//THIS^.bReset := TRUE;
		THIS^.eState := E_StateTerminal.RESETING;
		
	(* Reset all control variables *)
	E_StateTerminal.RESETING:
		//THIS^.bReset := FALSE;
		THIS^.eState := E_StateTerminal.INIT;	
		
	(* Enable terminal if ready *)
	E_StateTerminal.INIT:			
		THIS^.eState := E_StateTerminal.READY;

	(* Terminal is ready *)
	E_StateTerminal.READY:
		fbFeedback.Done := TRUE;
		
		
	(* Terminal is triggering *)
	E_StateTerminal.TRIGGERING:
		//WaitForTriggerDone:
		IF (F_GetCurDcTaskTime64()(*1ns*) >= THIS^.nStartTime) THEN
			THIS^.eState := E_StateTerminal.READY;
		 END_IF
			
	
	(* Error occured *)	
	E_StateTerminal.ERROR:
		fbFeedback.HR := E_FAIL;
		IF NOT THIS^.fbAlarmGeneral.bRaised THEN
			THIS^.fbAlarmGeneral.Raise(0);	
		END_IF
		
		IF (THIS^.fbAlarmGeneral.eConfirmationState = TcEventConfirmationState.Confirmed) THEN
			THIS^.Reset();			
		END_IF			
END_CASE

(* Timeout if an actingstate is to long active *)
fbTimeout.IN := (THIS^.eState = E_StateTerminal.INIT) OR (THIS^.eState = E_StateTerminal.RESETING) OR (THIS^.eState = E_StateTerminal.TRIGGERING);
fbTimeout.PT := T#5S;
fbTimeout();
IF fbTimeout.Q THEN
	THIS^.eState := E_StateTerminal.ERROR;
END_IF
END_METHOD

END_FUNCTION_BLOCK

// COMPONENTs/CameraTriggerController/EtherCAT Timestamp trigger/I_SwTimestamp_Mode
INTERFACE I_SwTimestamp_Mode EXTENDS __SYSTEM.IQueryInterface

METHOD PUBLIC Trigger : HRESULT
VAR_INPUT
	//The data type T_DCTIME64 represents the distributed clock system time (abbreviated as DC time) as a linear 64-bit integer value. 
	//The time is expressed in nanoseconds since 1/1/2000 UTC. The smallest unit is a nanosecond.
	//F_GetCurDcTickTime64()
	nDCTimeStamp	: T_DCTIME64;
END_VAR
END_METHOD

{attribute 'monitoring' := 'call'}
// The given trigger time is delayed by this value. E.g. to wait for the maximum lighting value before taking a picture  [in 1ns]
PROPERTY TriggerDelay_1ns : UDINT
GET
END_GET
SET
END_SET
END_PROPERTY

END_INTERFACE

// COMPONENTs/CameraTriggerController/EtherCAT Timestamp trigger/FB_EtherCAT_Trigger_old
{attribute 'no_explicit_call' := 'Do not call the body - Stick to OOP'}
FUNCTION_BLOCK FB_EtherCAT_Trigger_old EXTENDS FB_CameraTriggerController_Base IMPLEMENTS I_SwTimestamp_Mode
VAR
	nStartTime 				AT %Q*	: T_DCTIME64;			// Trigger time stamp
	nActivate				AT %Q*	: USINT; 				// 0 -> 3 use new time in terminal
	
	{attribute 'hide'}
	nTriggerDelay 			: UDINT := 0;					// The given trigger time is delayed by this value. E.g. to wait for the maximum lighting value before taking a picture  [in 100ns]
	
	{attribute 'hide'}
	eState					: E_StateTerminal;				// Current terminal state
END_VAR

{attribute 'monitoring' := 'call'}
PROPERTY Operational : BOOL
GET
Operational := (THIS^.eState = E_StateTerminal.READY) OR (THIS^.eState = E_StateTerminal.TRIGGERING);
END_GET
END_PROPERTY

METHOD PUBLIC Reset : HRESULT
VAR_INPUT
END_VAR
IF THIS^.eState = E_StateTerminal.ERROR THEN
	fbFeedback.ActiveCommand := 'Reset';
	fbFeedback.Busy := TRUE;	

	THIS^.eState := E_StateTerminal.RESET;
END_IF
END_METHOD

{attribute 'monitoring' := 'call'}
PROPERTY PUBLIC State : E_StateTerminal
GET
State := THIS^.eState;
END_GET
END_PROPERTY

METHOD PUBLIC Trigger : HRESULT
VAR_INPUT
	//The data type T_DCTIME64 represents the distributed clock system time (abbreviated as DC time) as a linear 64-bit integer value. 
	//The time is expressed in nanoseconds since 1/1/2000 UTC. The smallest unit is a nanosecond.
	//F_GetCurDcTickTime64()
	nDCTimeStamp	: T_DCTIME64;
END_VAR
(* Check if the trigger is minimum 3 EtherCat cycles in future *)
IF (nDCTimeStamp + THIS^.nTriggerDelay) < THIS^.NextPossibleTriggerTime THEN
	Trigger := E_FAIL;
	RETURN;
END_IF

(* Check if not in wrong state *)
IF NOT (THIS^.eState = E_StateTerminal.READY) THEN
	Trigger := E_FAIL;
	RETURN;
END_IF

fbFeedback.ActiveCommand := 'Trigger';
fbFeedback.Busy := TRUE;	


THIS^.nStartTime := nDCTimeStamp + THIS^.nTriggerDelay;
THIS^.nActivate := 3; (*Activate*)

THIS^.eState := E_StateTerminal.TRIGGERING;
Trigger := S_OK;
END_METHOD

{attribute 'monitoring' := 'call'}
// The given trigger time is delayed by this value. E.g. to wait for the maximum lighting value before taking a picture  [in 1ns]
PROPERTY TriggerDelay_1ns : UDINT
GET
TriggerDelay_1ns := THIS^.nTriggerDelay;
END_GET
SET
THIS^.nTriggerDelay := TriggerDelay_1ns;
END_SET
END_PROPERTY

METHOD PUBLIC Update : HRESULT
VAR_INST
	{attribute 'hide'}
	fbTimeout : TON;
END_VAR
(* Handle terminal state machine *)
CASE THIS^.eState OF
	(* Reset all control variables *)
	E_StateTerminal.RESET:
		//THIS^.bReset := TRUE;
		THIS^.eState := E_StateTerminal.RESETING;
		
	(* Reset all control variables *)
	E_StateTerminal.RESETING:
		//THIS^.bReset := FALSE;
		THIS^.eState := E_StateTerminal.INIT;	
		
	(* Enable terminal if ready *)
	E_StateTerminal.INIT:			
		THIS^.eState := E_StateTerminal.READY;

	(* Terminal is ready *)
	E_StateTerminal.READY:
		fbFeedback.Done := TRUE;
		THIS^.nActivate := 0;
		
		
	(* Terminal is triggering *)
	E_StateTerminal.TRIGGERING:
		//WaitForTriggerDone:
		IF (F_GetCurDcTaskTime64()(*1ns*) >= (THIS^.nStartTime)) THEN
			//Befor leave triggering, stay 1 cycle in Activate=0
			IF THIS^.nActivate = 0 THEN
				THIS^.eState := E_StateTerminal.READY;
			ELSE 
				THIS^.nActivate := 0;(*Deactivate*)
			END_IF

		 END_IF
			
	
	(* Error occured *)	
	E_StateTerminal.ERROR:
		fbFeedback.HR := E_FAIL;
		IF NOT THIS^.fbAlarmGeneral.bRaised THEN
			THIS^.fbAlarmGeneral.Raise(0);	
		END_IF
		
		IF (THIS^.fbAlarmGeneral.eConfirmationState = TcEventConfirmationState.Confirmed) THEN
			THIS^.Reset();			
		END_IF			
END_CASE

(* Timeout if an actingstate is to long active *)
fbTimeout.IN := (THIS^.eState = E_StateTerminal.INIT) OR (THIS^.eState = E_StateTerminal.RESETING) OR (THIS^.eState = E_StateTerminal.TRIGGERING);
fbTimeout.PT := T#5S;
fbTimeout();
IF fbTimeout.Q THEN
	THIS^.eState := E_StateTerminal.ERROR;
END_IF
END_METHOD

END_FUNCTION_BLOCK

// COMPONENTs/CameraTriggerController/GigE - Softwaretrigger/FB_GigeSoftwaretrigger
{attribute 'no_explicit_call' := 'Do not call the body - Stick to OOP'}
FUNCTION_BLOCK FB_GigeSoftwaretrigger EXTENDS FB_CameraTriggerController_Base IMPLEMENTS I_GigeSoftTrigger_Mode
VAR
	{attribute 'hide'}
	eState							: E_StateTerminal;		// Current terminal state
	nTimeNextTrigger : T_DCTIME64;
	nTriggerDelay : UDINT := 10;			// Delay between lighting and camera trigger [in 1ns]
	ipGigeCamera : I_GigEVision_Mode;
	
END_VAR

PROPERTY Duration_1us : UDINT
GET
END_GET
SET
END_SET
END_PROPERTY

PROPERTY GigeCamera : I_GigEVision_Mode
GET
GigeCamera := ipGigeCamera;
END_GET
SET
ipGigeCamera := GigeCamera;
END_SET
END_PROPERTY

METHOD PUBLIC Reset : HRESULT
VAR_INPUT
END_VAR
IF (THIS^.eState = E_StateTerminal.ERROR) THEN
	fbFeedback.ActiveCommand := 'Reset';
	fbFeedback.Busy := TRUE;	

	THIS^.eState := E_StateTerminal.RESET;
END_IF
END_METHOD

METHOD Trigger : HRESULT
VAR_INPUT
	//The data type T_DCTIME64 represents the distributed clock system time (abbreviated as DC time) as a linear 64-bit integer value. 
	//The time is expressed in nanoseconds since 1/1/2000 UTC. The smallest unit is a nanosecond.
	//F_GetCurDcTickTime64()
	nDCTimeStamp	: T_DCTIME64;
END_VAR
THIS^.nTimeNextTrigger := nDCTimeStamp;
THIS^.eState := E_StateTerminal.TRIGGERING;

fbFeedback.ActiveCommand := 'Trigger';
fbFeedback.Busy := TRUE;	



Trigger := S_OK;
END_METHOD

{attribute 'monitoring' := 'call'}
// The given trigger time is delayed by this value. E.g. to wait for the maximum lighting value before taking a picture  [in 1ns]
PROPERTY TriggerDelay_1ns : UDINT
GET
TriggerDelay_1ns := THIS^.nTriggerDelay;
END_GET
SET
THIS^.nTriggerDelay := TriggerDelay_1ns;
END_SET
END_PROPERTY

METHOD PUBLIC Update : HRESULT
VAR_INST

END_VAR
VAR
	
	fbTaskInfo		 : PlcTaskSystemInfo;
END_VAR
IF THIS^.ipGigeCamera = 0 THEN
	THIS^.eState := E_StateTerminal.ERROR;
END_IF


(* Handle terminal state machine *)
CASE THIS^.eState OF
	(* Reset all control variables *)
	E_StateTerminal.RESET:
		THIS^.eState := E_StateTerminal.RESETING;
		
	(* Reset all control variables *)
	E_StateTerminal.RESETING:
		THIS^.eState := E_StateTerminal.INIT;	
		
	(* Enable terminal if ready *)
	E_StateTerminal.INIT:			
		THIS^.eState := E_StateTerminal.READY;
	
	(* Terminal is ready *)
	E_StateTerminal.READY:
		fbFeedback.Done := TRUE;	
		
	(* Terminal is triggering *)
	E_StateTerminal.TRIGGERING:
		IF (F_GetCurDcTaskTime64()  >=   (THIS^.nTimeNextTrigger - TO_ULINT(THIS^.nTriggerDelay))) THEN
			THIS^.ipGigeCamera.Softtrigger();
			THIS^.eState := E_StateTerminal.READY;
		END_IF
	
	(* Error occured *)	
	E_StateTerminal.ERROR:
		fbFeedback.HR := E_FAIL;
		;

END_CASE
END_METHOD

END_FUNCTION_BLOCK

// COMPONENTs/CameraTriggerController/GigE - Softwaretrigger/I_GigeSoftTrigger_Mode
INTERFACE I_GigeSoftTrigger_Mode EXTENDS __SYSTEM.IQueryInterface

PROPERTY GigeCamera : I_GigEVision_Mode
GET
END_GET
SET
END_SET
END_PROPERTY

METHOD Trigger : HRESULT
VAR_INPUT
	//The data type T_DCTIME64 represents the distributed clock system time (abbreviated as DC time) as a linear 64-bit integer value. 
	//The time is expressed in nanoseconds since 1/1/2000 UTC. The smallest unit is a nanosecond.
	//F_GetCurDcTickTime64()
	nDCTimeStamp	: T_DCTIME64;
END_VAR
END_METHOD

{attribute 'monitoring' := 'call'}
PROPERTY TriggerDelay_1ns : UDINT
GET
END_GET
SET
END_SET
END_PROPERTY

END_INTERFACE

// COMPONENTs/ImageProvider/Camera/I_GigEVision_Mode
INTERFACE I_GigEVision_Mode

{attribute 'monitoring' := 'call'}
PROPERTY Exposure_1us : UDINT
GET
END_GET
SET
END_SET
END_PROPERTY

METHOD PUBLIC Softtrigger : HRESULT
END_METHOD

END_INTERFACE

// COMPONENTs/IlluminationController/EL2595 - 1Ch. LED output timestamp/FB_EL2595
{attribute 'no_explicit_call' := 'Do not call the body - Stick to OOP'}
FUNCTION_BLOCK FB_EL2595 EXTENDS FB_IlluminationController_Base IMPLEMENTS I_IlluminationSingleOutput_Mode
VAR
	(*DOX Control*)
	bOutput					AT %Q* 	: BOOL;					// Desired State of Output
	bReset					AT %Q*	: BOOL;					// Terminal reset
	
	(*DC Sync*)
	nStartTime 				AT %Q*	: T_DCTIME64;			// Trigger time stamp
	nActivate				AT %Q*	: USINT; 				// 0 -> 3 use new time in terminal
	
	(*DOX Status*)
	bReadyToActivate		AT %I*	: BOOL := FALSE;		// Terminal ready
	bWarning				AT %I*	: BOOL := FALSE;		// Terminal has warning
	bError					AT %I*	: BOOL := FALSE;		// Terminal has error
	
	(*DC Feedback*)
	nDCFeedback				AT %I*  : USINT := 0;			// Feedback of outputchanel
	

	nImpulseLength 			AT %Q* 	: UDINT := 20000;   	// Impulse length of the lighting period [in 1us]
	nTriggerDelay 			AT %Q* 	: UDINT := 10;			// Delay between lighting and camera trigger [in 100ns]

	{attribute 'hide'}
	eState					: E_StateTerminal;				// Current terminal state
	eTriggerSubState		:(SEQ_WirteTime, SEQ_Activate, SEQ_WaitForFeedback, SEQ_Done); //setting the trigger takes several Ethercat cycles
END_VAR

{attribute 'monitoring' := 'call'}
//Module already has a task - already a trigger active
PROPERTY Busy : BOOL
GET
Busy := (THIS^.eState = E_StateTerminal.TRIGGERING);
END_GET
END_PROPERTY

{attribute 'monitoring' := 'call'}
PROPERTY Duration_1us : UDINT
GET
Duration_1us := THIS^.nImpulseLength;
END_GET
SET
THIS^.nImpulseLength := Duration_1us;
END_SET
END_PROPERTY

{attribute 'monitoring' := 'call'}
PROPERTY Operational : BOOL
GET
Operational := (THIS^.eState = E_StateTerminal.READY) OR (THIS^.eState = E_StateTerminal.TRIGGERING);
END_GET
END_PROPERTY

METHOD PUBLIC Reset : HRESULT
VAR_INPUT
END_VAR
IF NOT THIS^.Operational THEN
	THIS^.eState := E_StateTerminal.RESET;
END_IF
END_METHOD

{attribute 'monitoring' := 'call'}
PROPERTY PUBLIC State : E_StateTerminal
GET
State := THIS^.eState;
END_GET
END_PROPERTY

METHOD PUBLIC Trigger : HRESULT
VAR_INPUT
	//The data type T_DCTIME64 represents the distributed clock system time (abbreviated as DC time) as a linear 64-bit integer value. 
	//The time is expressed in nanoseconds since 1/1/2000 UTC. The smallest unit is a nanosecond.
	//F_GetCurDcTickTime64()
	nDCTimeStamp	: T_DCTIME64;
END_VAR
(* Check if the trigger is minimum 3 EtherCat cycles in future *)
IF nDCTimeStamp < THIS^.NextPossibleTriggerTime  THEN
	Trigger := E_FAIL;
	RETURN;
END_IF

(* Check if not in wrong state *)
IF NOT (THIS^.eState = E_StateTerminal.READY) THEN
	Trigger := E_FAIL;
	RETURN;
END_IF




THIS^.nStartTime := nDCTimeStamp;
THIS^.bOutput := TRUE;
THIS^.nActivate := 0;

THIS^.eTriggerSubState := SEQ_WirteTime;
THIS^.eState := E_StateTerminal.TRIGGERING;
Trigger := S_OK;
END_METHOD

METHOD PUBLIC Update : HRESULT
VAR_INST
	fbTimeout : TON;
END_VAR
(* Check for terminal errors *)
IF THIS^.bError AND NOT (THIS^.eState = E_StateTerminal.RESET) THEN 
	THIS^.eState := E_StateTerminal.ERROR;
END_IF

(* Handle terminal state machine *)
CASE THIS^.eState OF
	(* Reset all control variables *)
	E_StateTerminal.RESET:
		THIS^.bReset := TRUE;
		THIS^.eState := E_StateTerminal.RESETING;
		
	(* Reset all control variables *)
	E_StateTerminal.RESETING:
		THIS^.bReset := FALSE;
		THIS^.eState := E_StateTerminal.INIT;	
		
	(* Enable terminal if ready *)
	E_StateTerminal.INIT:			
		IF THIS^.bReadyToActivate THEN
			THIS^.bReset := FALSE;
			THIS^.fbAlarmGeneral.Clear(0, TRUE);
			THIS^.eState := E_StateTerminal.READY;
		END_IF
	
	(* Terminal is ready *)
	E_StateTerminal.READY:
		THIS^.nStartTime := 0;
		THIS^.bOutput := FALSE;
		THIS^.nActivate := 0;

	(* Terminal is triggering *)
	E_StateTerminal.TRIGGERING:
		CASE eTriggerSubState OF
			SEQ_WirteTime:
				//Wirte TimeStamp, Output and Activate=0 in .Trigger()
				//The next commands are allowed only in the next Ethercat cycle
				eTriggerSubState := SEQ_Activate;
				
			SEQ_Activate:
				// Activate new time
				THIS^.nActivate := 3;
				eTriggerSubState := SEQ_WaitForFeedback;
				
			SEQ_WaitForFeedback:
				// Trigger is done and PulsOffTime is done
				IF ((F_GetCurDcTaskTime64()(*100ns*) > THIS^.nStartTime) AND THIS^.bReadyToActivate) THEN
					THIS^.nActivate := 0;
					eTriggerSubState := SEQ_Done;
					//Ready for next Trigger
					THIS^.eState := E_StateTerminal.READY;
				END_IF

			SEQ_Done:
			;
		END_CASE
	
	
	(* Error occured *)	
	E_StateTerminal.ERROR:
		IF NOT THIS^.fbAlarmGeneral.bRaised THEN
			THIS^.fbAlarmGeneral.Raise(0);	
		END_IF
		
		IF (THIS^.fbAlarmGeneral.eConfirmationState = TcEventConfirmationState.Confirmed) THEN
			THIS^.Reset();			
		END_IF			
END_CASE

(* Timeout if an state is to long active *)
fbTimeout.IN := (THIS^.eState = E_StateTerminal.INIT) OR (THIS^.eState = E_StateTerminal.RESETING) OR (THIS^.eState = E_StateTerminal.TRIGGERING);
fbTimeout.PT := T#5S;
fbTimeout();
IF fbTimeout.Q THEN
	THIS^.eState := E_StateTerminal.ERROR;
END_IF
END_METHOD

END_FUNCTION_BLOCK

// COMPONENTs/IlluminationController/FB_IlluminationController_Base
{attribute 'no_explicit_call' := 'Do not call the body - Stick to OOP'}
FUNCTION_BLOCK ABSTRACT FB_IlluminationController_Base EXTENDS FB_CH_Object IMPLEMENTS I_IlluminationController_Base
VAR
	ipVisionSystem		: I_VisionSystem;			// Interface to "Owner" of this module. Visionsystem
	fbAlarmGeneral 		: FB_TcAlarm;			// Terminal general alarm
END_VAR

{attribute 'monitoring' := 'call'}
//Module already has a task - already a trigger active
PROPERTY ABSTRACT Busy : BOOL
GET
END_GET
END_PROPERTY

{attribute 'monitoring' := 'call'}
PROPERTY NextPossibleTriggerTime : T_DCTIME64
GET
VAR
	nEtherCatCycles 	: UINT;	
END_VAR
//If attribute 'TcCallAfterOutputUpdate' is set, it takes 1 cycle more to send timestamp to hardware
IF TwinCAT_SystemInfoVarList._TaskInfo[THIS^.TaskIndex].InCallAfterOutputUpdate THEN
	nEtherCatCycles := 3;
ELSE
	nEtherCatCycles := 2;
END_IF


NextPossibleTriggerTime := F_GetCurDcTaskTime64()(*1ns*) + (THIS^.ipVisionSystem.TaskCycleTimeNs(*1ns*) * nEtherCatCycles (*Cycles*)) + 300_000(*300us(determined by testing)*);
END_GET
END_PROPERTY

{attribute 'monitoring' := 'call'}
PROPERTY ABSTRACT Operational : BOOL
GET
END_GET
END_PROPERTY

METHOD ABSTRACT Reset : HRESULT
END_METHOD

METHOD SetParent
VAR_INPUT
	ipVisionSystem  : I_VisionSystem;
END_VAR
THIS^.ipVisionSystem := ipVisionSystem;
END_METHOD

{attribute 'monitoring' := 'call'}
PROPERTY ABSTRACT State : E_StateTerminal
GET
END_GET
END_PROPERTY

METHOD ABSTRACT Trigger : HRESULT
VAR_INPUT
	//The data type T_DCTIME64 represents the distributed clock system time (abbreviated as DC time) as a linear 64-bit integer value. 
	//The time is expressed in nanoseconds since 1/1/2000 UTC. The smallest unit is a nanosecond.
	//F_GetCurDcTickTime64()
	nDCTimeStamp	: T_DCTIME64;
END_VAR
END_METHOD

END_FUNCTION_BLOCK

// COMPONENTs/IlluminationController/SingleOutput/I_IlluminationSingleOutput_Mode
INTERFACE I_IlluminationSingleOutput_Mode

{attribute 'monitoring' := 'call'}
PROPERTY Duration_1us : UDINT
GET
END_GET
SET
END_SET
END_PROPERTY

METHOD  Trigger : HRESULT
VAR_INPUT
	//The data type T_DCTIME64 represents the distributed clock system time (abbreviated as DC time) as a linear 64-bit integer value. 
	//The time is expressed in nanoseconds since 1/1/2000 UTC. The smallest unit is a nanosecond.
	//F_GetCurDcTickTime64()
	nDCTimeStamp	: T_DCTIME64;
END_VAR
END_METHOD

END_INTERFACE

// COMPONENTs/IlluminationController/SingleOutput/FB_IlluminationSingleOutput
FUNCTION_BLOCK FB_IlluminationSingleOutput EXTENDS FB_IlluminationController_Base
VAR
	bTrigger 			AT %Q* 	: BOOL;			// Trigger for lighting
	
	nImpulseLength 		: UINT;   				// Impulse length of the lighting period [ms]
	eState				: E_StateTerminal  := E_StateTerminal.READY;		// Current terminal state
	
	fbTriggerOffDelay	: TOF;
END_VAR

{attribute 'monitoring' := 'call'}
//Module already has a task - already a trigger active
PROPERTY Busy : BOOL
GET
Busy := THIS^.eState = E_StateTerminal.TRIGGERING;
END_GET
END_PROPERTY

METHOD Configure : HRESULT
VAR_INPUT

END_VAR
END_METHOD

METHOD FB_init : BOOL
VAR_INPUT
	bInitRetains : BOOL; // if TRUE, the retain variables are initialized (warm start / cold start)
	bInCopyCode : BOOL;  // if TRUE, the instance afterwards gets moved into the copy code (online change)
	
	nImpulseLength 	: UINT;   	// Impulse length of the lighting period [ms]
END_VAR
VAR_INST
	{attribute 'hide'}
	bFBInitCalledOnce : BOOL; //Do the following code once during start up and not during onlinechange
END_VAR
//Do the following code once during start up and not during onlinechange
IF NOT bFBInitCalledOnce THEN 
	

	THIS^.nImpulseLength 	:= nImpulseLength; 	 	


END_IF

bFBInitCalledOnce := TRUE;
END_METHOD

METHOD Initialize : HRESULT
VAR
	hr : HRESULT;
END_VAR
hr := SUPER^.Initialize();

THIS^.eState := E_StateTerminal.READY;
THIS^.fbTriggerOffDelay.PT := UINT_TO_TIME(THIS^.nImpulseLength);

Initialize := hr;
END_METHOD

{attribute 'monitoring' := 'call'}
PROPERTY Operational : BOOL
GET
Operational := (THIS^.eState = E_StateTerminal.READY) OR (THIS^.eState = E_StateTerminal.TRIGGERING);
END_GET
END_PROPERTY

METHOD  Reset : HRESULT
Reset := S_OK;
END_METHOD

{attribute 'monitoring' := 'call'}
PROPERTY PUBLIC State : E_StateTerminal
GET

State := THIS^.eState;
END_GET
END_PROPERTY

METHOD  Trigger : HRESULT
VAR_INPUT
	//The data type T_DCTIME64 represents the distributed clock system time (abbreviated as DC time) as a linear 64-bit integer value. 
	//The time is expressed in nanoseconds since 1/1/2000 UTC. The smallest unit is a nanosecond.
	//F_GetCurDcTickTime64()
	nDCTimeStamp	: T_DCTIME64;
END_VAR
(* Check if the trigger is minimum 3 EtherCat cycles in future *)
IF nDCTimeStamp < THIS^.NextPossibleTriggerTime  THEN
	Trigger := E_FAIL;
	RETURN;
END_IF

(* The trigger methode can be called in each state. 
Is the output is already set, the off-timer is resetet *)

THIS^.fbTriggerOffDelay.IN := TRUE;;
Trigger := S_OK;
END_METHOD

METHOD PUBLIC Update : HRESULT
(* The trigger methode call be called in each state. 
Is the output is already set, the off-timer is resetet *)

(* Handle terminal state machine *)
CASE THIS^.eState OF
	(* Terminal is ready *)
	E_StateTerminal.READY:
		;		
	(* Terminal is triggering *)
	E_StateTerminal.TRIGGERING:
		;
END_CASE

THIS^.fbTriggerOffDelay();
THIS^.fbTriggerOffDelay.IN := FALSE;

//Set Output
THIS^.bTrigger := THIS^.fbTriggerOffDelay.Q;

//Set State
IF THIS^.bTrigger THEN
	THIS^.eState := E_StateTerminal.TRIGGERING;
ELSE	
	THIS^.eState := E_StateTerminal.READY;
END_IF
END_METHOD

END_FUNCTION_BLOCK

// COMPONENTs/IlluminationController/VIx2000/FB_VIx2000
{attribute 'no_explicit_call' := 'Do not call the body - Stick to OOP'}
FUNCTION_BLOCK FB_VIx2000 EXTENDS FB_IlluminationController_Base IMPLEMENTS I_IlluminationController_Base, I_VIx2000_Mode
VAR
	DeviceInputs 	 		AT %I* 	: ST_VIx2000_InDevice;
	DeviceOutputs			AT %Q*	: ST_VIx2000_OutDevice;		
	Pulse_DC_Outputs		AT %Q*	: ST_VIx2000_Pulse;		
	ChannelOrange 			AT %Q*	: ST_VIx2000_Channel;
	ChannelGreen 			AT %Q*	: ST_VIx2000_Channel;
	ChannelBlue 			AT %Q*	: ST_VIx2000_Channel;
	ChannelInfrared 		AT %Q*	: ST_VIx2000_Channel;
	
	
	{attribute 'hide'}
	bInitDone 						: BOOL;
	{attribute 'hide'}	
	eState							: E_VIx2000_Status;
	{attribute 'hide'}	
	nDuration_1us					: UDINT := 100_000; //Puls duration
	{attribute 'hide'}
	nSwitchOnCounterOnTrigger		: UDINT;				// Old operation counter as reference
	{attribute 'hide'}
	fbFeedBackTrigger 				: FB_CH_Feedback(THIS^.fbSourceInfo);
END_VAR
VAR CONSTANT
	N_MAX_BRIGHTNESS : UINT := 511;
END_VAR

{attribute 'monitoring' := 'call'}
//Module already has a task - already a trigger active
PROPERTY Busy : BOOL
GET
Busy := (THIS^.eState = E_VIx2000_Status.TRIGGERING);
END_GET
END_PROPERTY

METHOD Configure : HRESULT
VAR_INPUT
	nOrange 	: UINT(0..N_MAX_BRIGHTNESS);
	nGreen 		: UINT(0..N_MAX_BRIGHTNESS);
	nBlue 		: UINT(0..N_MAX_BRIGHTNESS);
	nInfrared 	: UINT(0..N_MAX_BRIGHTNESS);
	nDuration_1us : UDINT; //Duration of pulse
END_VAR
THIS^.ChannelOrange.nBrightness := LIMIT(0, nOrange, N_MAX_BRIGHTNESS);
THIS^.ChannelGreen.nBrightness := LIMIT(0, nGreen, N_MAX_BRIGHTNESS);
THIS^.ChannelBlue.nBrightness := LIMIT(0, nBlue, N_MAX_BRIGHTNESS);
THIS^.ChannelInfrared.nBrightness := LIMIT(0, nInfrared, N_MAX_BRIGHTNESS);

THIS^.ChannelOrange.nDuration_1us := nDuration_1us;
THIS^.ChannelGreen.nDuration_1us := nDuration_1us;
THIS^.ChannelBlue.nDuration_1us := nDuration_1us;
THIS^.ChannelInfrared.nDuration_1us := nDuration_1us;

THIS^.nDuration_1us := nDuration_1us;
END_METHOD

{attribute 'monitoring' := 'call'}
PROPERTY Duration_1us : UDINT
GET
Duration_1us := THIS^.nDuration_1us;
END_GET
SET
THIS^.nDuration_1us := Duration_1us;

THIS^.ChannelOrange.nDuration_1us := Duration_1us;
THIS^.ChannelGreen.nDuration_1us := Duration_1us;
THIS^.ChannelBlue.nDuration_1us := Duration_1us;
THIS^.ChannelInfrared.nDuration_1us := Duration_1us;
END_SET
END_PROPERTY

{attribute 'monitoring' := 'call'}
PROPERTY Enable : BOOL
GET
Enable := THIS^.DeviceOutputs.bEnable;
END_GET
END_PROPERTY

METHOD Initialize : HRESULT
VAR
	ipChObject 			: I_CH_OBJECT;
	hr: HRESULT;
END_VAR
hr := SUPER^.Initialize();

//Init some default data 
Configure(
	nOrange:= 50, 
	nGreen:= 50, 
	nBlue:= 50, 
	nInfrared:= 50, 
	nDuration_1us:= 10_000);

IF CheckOk(hr) THEN
	THIS^.bInitDone := TRUE;
END_IF

Initialize := hr;
END_METHOD

{attribute 'monitoring' := 'call'}
PROPERTY Operational : BOOL
GET
Operational := (THIS^.eState = E_VIx2000_Status.READY) OR (THIS^.eState = E_VIx2000_Status.TRIGGERING);
END_GET
END_PROPERTY

METHOD PUBLIC Reset : HRESULT
VAR_INPUT
END_VAR
IF NOT THIS^.Operational THEN
	 THIS^.eState := E_VIx2000_Status.RESET;
END_IF
END_METHOD

{attribute 'monitoring' := 'call'}
PROPERTY PUBLIC State : E_StateTerminal
GET
CASE THIS^.eState OF
	E_VIx2000_Status.INIT:
		State := E_StateTerminal.INIT;
		
	E_VIx2000_Status.READY:
		State := E_StateTerminal.READY;
		
	E_VIx2000_Status.TRIGGERING:
		State := E_StateTerminal.TRIGGERING;
		
	E_VIx2000_Status.ERROR:
		State := E_StateTerminal.ERROR;
		
	E_VIx2000_Status.RESET:
		State := E_StateTerminal.RESET;
		
	E_VIx2000_Status.RESETING:	
		State := E_StateTerminal.RESETING;
END_CASE
END_GET
END_PROPERTY

METHOD Trigger : HRESULT
VAR_INPUT
	//The data type T_DCTIME64 represents the distributed clock system time (abbreviated as DC time) as a linear 64-bit integer value. 
	//The time is expressed in nanoseconds since 1/1/2000 UTC. The smallest unit is a nanosecond.
	//F_GetCurDcTickTime64()
	nDCTimeStamp : T_DCTIME64;
END_VAR
(* Check if the trigger is minimum 3 EtherCat cycles in future *)
IF nDCTimeStamp < THIS^.NextPossibleTriggerTime THEN
	Trigger := E_FAIL;
	RETURN;
END_IF



IF (THIS^.eState = E_VIx2000_Status.READY) THEN
	THIS^.nSwitchOnCounterOnTrigger := THIS^.DeviceInputs.nSwitch_on_counter;
	THIS^.Pulse_DC_Outputs.nTimestamp 	:= nDCTimeStamp;
	THIS^.Pulse_DC_Outputs.nFlashDelay 	:= 0;

	THIS^.eState := E_VIx2000_Status.TRIGGERING;
	
	THIS^.fbFeedbackTrigger.hr := S_OK;
ELSE
	THIS^.fbFeedbackTrigger.hr := E_FAIL;
END_IF

Trigger := THIS^.fbFeedbackTrigger.hr;
END_METHOD

METHOD Update : HRESULT
VAR
	bNewCounterValue : BOOL;
END_VAR
VAR_INST
	{attribute 'hide'}
	nSwitchOnCounterShouldValue : UDINT;
	{attribute 'hide'}
	nSwitchOnCounterLastCycle : UDINT;
	{attribute 'hide'}
	fbTimeOutNoReactionToTrigger : TON;
	{attribute 'hide'}
	fbStateTimeout : TON;
	{attribute 'hide'}
	fbTimeoutAlarm : FB_TcAlarm;
	{attribute 'hide'}
	fbAlarmNoReactionToTrigger : FB_TcAlarm;
	{attribute 'hide'}
	eStateOld : E_VIx2000_Status;
END_VAR
(* Check for terminal errors *)
IF THIS^.DeviceInputs.bError AND NOT ((THIS^.eState = E_VIx2000_Status.RESET) OR (THIS^.eState = E_VIx2000_Status.RESETING))THEN 
	THIS^.eState := E_VIx2000_Status.ERROR;
END_IF

(* Handle terminal state machine *)
CASE THIS^.eState OF
	(* Reset all control variables *)
	E_VIx2000_Status.RESET:
		THIS^.DeviceOutputs.bEnable := FALSE;
		THIS^.DeviceOutputs.bReset := FALSE;
		THIS^.Pulse_DC_Outputs.nTimestamp := 0;		
		THIS^.Pulse_DC_Outputs.nTimestamp := 0;	
		fbTimeoutAlarm.Clear(0,0);	
		fbAlarmNoReactionToTrigger.Clear(0,0);
		THIS^.fbFeedbackTrigger.HR := S_OK;
		
		THIS^.eState := E_VIx2000_Status.RESETING;
		
	(* Reset all control variables *)
	E_VIx2000_Status.RESETING:
		THIS^.DeviceOutputs.bEnable := FALSE;
		THIS^.DeviceOutputs.bReset := TRUE;
		THIS^.eState := E_VIx2000_Status.INIT;
	
	(* Enable terminal if ready *)
	E_VIx2000_Status.INIT:			
		THIS^.DeviceOutputs.bEnable := TRUE;
		THIS^.DeviceOutputs.bReset := FALSE;
		IF THIS^.DeviceInputs.bReady THEN
			THIS^.fbAlarmGeneral.Clear(0, TRUE);
			nSwitchOnCounterShouldValue := THIS^.DeviceInputs.nSwitch_on_counter;
			THIS^.eState := E_VIx2000_Status.READY;
		END_IF
	
	(* Terminal is ready *)
	E_VIx2000_Status.READY:
		;
		
	(* Terminal is triggering *)
	E_VIx2000_Status.TRIGGERING:
	IF VisionParameterlist.ILLUMINATION_WAIT_FOR_TRIGGER_FEEDBACK THEN
		//Wait - timeout if no change
		IF (THIS^.nSwitchOnCounterOnTrigger +1) = THIS^.DeviceInputs.nSwitch_on_counter THEN
			THIS^.eState := E_VIx2000_Status.READY;
		END_IF
	ELSE
		//Do not wait
		IF (F_GetCurDcTaskTime64()  >=  THIS^.Pulse_DC_Outputs.nTimestamp)  THEN
			nSwitchOnCounterShouldValue := nSwitchOnCounterShouldValue + 1;
			THIS^.eState := E_VIx2000_Status.READY;
		END_IF
	END_IF

	
	(* Error occured *)	
	E_VIx2000_Status.ERROR:
		IF NOT THIS^.fbAlarmGeneral.bRaised THEN
			THIS^.fbAlarmGeneral.Raise(0);	
		END_IF
		
		IF (THIS^.fbAlarmGeneral.eConfirmationState = TcEventConfirmationState.Confirmed) THEN
			THIS^.Reset();			
		END_IF			
END_CASE

(* Timeout if an state is to long active *)
fbStateTimeout.IN := (THIS^.eState = eStateOld) AND (THIS^.eState = E_VIx2000_Status.INIT) OR (THIS^.eState = E_VIx2000_Status.RESETING) OR (THIS^.eState = E_VIx2000_Status.TRIGGERING);
eStateOld := THIS^.eState;
fbStateTimeout.PT := T#5S;
fbStateTimeout();
IF fbStateTimeout.Q THEN
	//Raise TC3-Eventlogger Alarm
	IF NOT fbTimeOutAlarm.bRaised THEN
		fbTimeoutAlarm.CreateEx(stEventEntry := TC_EVENTS.CHALET_Vision_Events.TimeOut, bWithConfirmation := FALSE, ipSourceInfo := THIS^.fbSourceInfo);
		fbTimeoutAlarm.ipArguments.AddStringByValue(TO_STRING(THIS^.eState));
		fbTimeoutAlarm.Raise(0);
	END_IF
	
	//Change in alarm state
	THIS^.eState := E_VIx2000_Status.ERROR;
END_IF


//Check that the lighting reacts to the trigger signal within the given time and increments its switch-on counter
IF NOT VisionParameterlist.ILLUMINATION_WAIT_FOR_TRIGGER_FEEDBACK THEN
	bNewCounterValue := nSwitchOnCounterLastCycle <> THIS^.DeviceInputs.nSwitch_on_counter;
	nSwitchOnCounterLastCycle := THIS^.DeviceInputs.nSwitch_on_counter;
	fbTimeOutNoReactionToTrigger.IN := NOT bNewCounterValue AND (nSwitchOnCounterShouldValue <> THIS^.DeviceInputs.nSwitch_on_counter);
	fbTimeOutNoReactionToTrigger.PT := T#5S;
	fbTimeOutNoReactionToTrigger();
	IF fbTimeOutNoReactionToTrigger.Q THEN
		//Raise TC3-Eventlogger Alarm
		IF NOT fbAlarmNoReactionToTrigger.bRaised THEN
			fbAlarmNoReactionToTrigger.CreateEx(stEventEntry := TC_EVENTS.CHALET_Vision_Events.NoReactionToTheTrigger, bWithConfirmation := FALSE, ipSourceInfo := THIS^.fbSourceInfo);
			fbAlarmNoReactionToTrigger.Raise(0);
			nSwitchOnCounterShouldValue := THIS^.DeviceInputs.nSwitch_on_counter;
		END_IF
		
		//Change in alarm state
		THIS^.eState := E_VIx2000_Status.ERROR;
	END_IF
END_IF
END_METHOD

END_FUNCTION_BLOCK

// COMPONENTs/IlluminationController/VIx2000/I_VIx2000_Mode
INTERFACE I_VIx2000_Mode

METHOD Configure : HRESULT
VAR_INPUT
	nOrange 	: UINT(0..511);
	nGreen 		: UINT(0..511);
	nBlue 		: UINT(0..511);
	nInfrared 	: UINT(0..511);
	nDuration_1us : UDINT;
END_VAR
END_METHOD

METHOD Trigger : HRESULT
VAR_INPUT
	//The data type T_DCTIME64 represents the distributed clock system time (abbreviated as DC time) as a linear 64-bit integer value. 
	//The time is expressed in nanoseconds since 1/1/2000 UTC. The smallest unit is a nanosecond.
	//F_GetCurDcTickTime64()
	nDCTimeStamp	: T_DCTIME64;
END_VAR
END_METHOD

END_INTERFACE

// COMPONENTs/ImageProvider/Base FB/FB_ImageProvider_Base
{attribute 'no_explicit_call' := 'Do not call the body - Stick to OOP'}
FUNCTION_BLOCK ABSTRACT FB_ImageProvider_Base EXTENDS FB_CH_Object IMPLEMENTS I_ImageProvider_Base
VAR      	
	{attribute 'hide'}							
    fbCrititcalSection : FB_IecCriticalSection;    						// Internal lock for test & set function                                  	
	{attribute 'hide'}														    		
	eState 				: ETcVnCameraState;		
	{attribute 'hide'}  						
	fbFeedback 			: FB_CH_Feedback(THIS^.fbSourceInfo); 
	{attribute 'hide'}
	fbAlarmOIDNotSet 	: FB_TcAlarm;									// Alarm due to source state	
	{attribute 'hide'}
	ipVisionSystem		: I_CH_Object;									// Interface to "Owner" of this module. Visionsystem
END_VAR

METHOD FB_init : BOOL
VAR_INPUT
	bInitRetains : BOOL; // if TRUE, the retain variables are initialized (warm start / cold start)
	bInCopyCode : BOOL;  // if TRUE, the instance afterwards gets moved into the copy code (online change)
END_VAR
VAR_INST
	{attribute 'hide'}
	bFBInitCalledOnce : BOOL; //Do the following code once during start up and not during onlinechange
END_VAR
//Do the following code once during start up and not during onlinechange
IF NOT bFBInitCalledOnce THEN 
	
	;

END_IF

bFBInitCalledOnce := TRUE;
END_METHOD

{attribute 'monitoring':='call'}
PROPERTY Feedback : I_CH_Feedback
GET
Feedback := THIS^.fbFeedback;
END_GET
END_PROPERTY

METHOD Initialize : HRESULT
Initialize := S_OK;
END_METHOD

{attribute 'monitoring' := 'call'}
PROPERTY PUBLIC Operational : BOOL
// Module started successfully and entered aquiring mode
GET
Operational := (eState = TCVN_CS_ACQUIRING) OR (eState = TCVN_CS_TRIGGERING);
END_GET
END_PROPERTY

METHOD ABSTRACT Reset : HRESULT
END_METHOD

METHOD SetParent
VAR_INPUT
	ipObject : I_CH_Object;
END_VAR
THIS^.ipVisionSystem := ipObject;
END_METHOD

{attribute 'monitoring' := 'call'}
PROPERTY ABSTRACT State : ETcVnCameraState
GET
END_GET
END_PROPERTY

METHOD ABSTRACT TryGetImage : HRESULT
VAR_INPUT
	stImageWithInfo : REFERENCE TO ST_ImageWithInfo;
END_VAR
END_METHOD

END_FUNCTION_BLOCK

// COMPONENTs/ImageProvider/Camera/FB_GigE_Beckhoff
{attribute 'no_explicit_call' := 'Do not call the body - Stick to OOP'}
FUNCTION_BLOCK FB_GigE_Beckhoff EXTENDS FB_ImageProvider_Base IMPLEMENTS I_GigEVision_Mode, I_GigEVision_Register_Connection
VAR
	// This FB provides the basic functionality to control a GigE Vision camera and access its calibration data.
	fbCamera 						: FB_VN_GevCameraControl;	

	{attribute 'hide'}
	bResetCommand	: BOOL;
END_VAR


VAR	
	//GigE-Camera-Register
	//Read/Write
	{attribute 'hide'}
	fbRegAcquisitionMode 		: FB_VnRegister_UDINT(ipCameraConnection := THIS^, nAddress := E_CameraRegisters_Beckhoff.pAcquisitionModeReg, nEndian := 0);
	{attribute 'hide'}
	fbRegTriggerMode	 		: FB_VnRegister_UDINT(ipCameraConnection := THIS^, nAddress := E_CameraRegisters_Beckhoff.pTriggerModeFrameStartReg, nEndian := 0);
	{attribute 'hide'}
	fbRegTriggerSource	 		: FB_VnRegister_UDINT(ipCameraConnection := THIS^, nAddress := E_CameraRegisters_Beckhoff.pTriggerSourceFrameStartReg, nEndian := 0);
	{attribute 'hide'}
	fbRegExposureTime	 		: FB_VnRegister_UDINT(ipCameraConnection := THIS^, nAddress := E_CameraRegisters_Beckhoff.pExposureTimeReg, nEndian := 0);
	{attribute 'hide'}
	fbRegDeviceDefaultState		: FB_VnRegister_UDINT(ipCameraConnection := THIS^, nAddress := E_CameraRegisters_Beckhoff.pDeviceDefaultStateReg, nEndian := 0);
	
	//Read only
	{attribute 'hide'}
	fbRegDeviceVendorName		: FB_VnRegister_Memory(ipCameraConnection := THIS^, nAddress := E_CameraRegisters_Beckhoff.DeviceVendorName, nLength := 32); //String	
	{attribute 'hide'}
	fbRegDeviceModelName	 	: FB_VnRegister_Memory(ipCameraConnection := THIS^, nAddress := E_CameraRegisters_Beckhoff.DeviceModelName, nLength := 32); //String	
	{attribute 'hide'}
	fbRegDeviceVersion	 		: FB_VnRegister_Memory(ipCameraConnection := THIS^, nAddress := E_CameraRegisters_Beckhoff.DeviceVersion, nLength := 32); //String	
	{attribute 'hide'}
	fbRegDeviceSerialNumber	 	: FB_VnRegister_Memory(ipCameraConnection := THIS^, nAddress := E_CameraRegisters_Beckhoff.DeviceSerialNumber, nLength := 16); //String	
	{attribute 'hide'}
	fbRegCurrentIPAddress	 	: FB_VnRegister_UDINT(ipCameraConnection := THIS^, nAddress := E_CameraRegisters_Beckhoff.BootStrap_IPAddress, nEndian := 0);  //T_IPv4AddrArr
	{attribute 'hide'}
	fbRegGevMACAddressHighWord	: FB_VnRegister_UDINT(ipCameraConnection := THIS^, nAddress := E_CameraRegisters_Beckhoff.pGevMACAddressHighWordReg, nEndian := 0);
	{attribute 'hide'}
	fbRegGevMACAddressLowWord	: FB_VnRegister_UDINT(ipCameraConnection := THIS^, nAddress := E_CameraRegisters_Beckhoff.pGevMACAddressLowWordReg, nEndian := 0);

	//List
	{attribute 'hide'}
	fbVnRegisterList 			: FB_CH_List;
END_VAR

{attribute 'monitoring' := 'call'}
PROPERTY DeviceDefaultState : E_DeviceDefaultState
GET
DeviceDefaultState := THIS^.fbRegDeviceDefaultState.Value;
END_GET
SET
IF THIS^.fbRegDeviceDefaultState.Value <> DeviceDefaultState THEN
 	//Set Camera from AQUIRING in OPENED - only on new value
	THIS^.fbCamera.StopAcquisition();
END_IF

THIS^.fbRegDeviceDefaultState.Value := DeviceDefaultState;
END_SET
END_PROPERTY

{attribute 'monitoring' := 'call'}
PROPERTY DeviceModeNamel : STRING
GET
fbRegDeviceModelName.ReadData(ADR(DeviceModeNamel));
END_GET
END_PROPERTY

{attribute 'monitoring' := 'call'}
PROPERTY DeviceSerialNumber : STRING
GET
fbRegDeviceSerialNumber.ReadData(ADR(DeviceSerialNumber));
END_GET
END_PROPERTY

{attribute 'monitoring' := 'call'}
PROPERTY DeviceVendorName : STRING
GET
fbRegDeviceVendorName.ReadData(ADR(DeviceVendorName));
END_GET
END_PROPERTY

{attribute 'monitoring' := 'call'}
PROPERTY DeviceVersion : STRING
GET
fbRegDeviceVersion.ReadData(ADR(DeviceVersion));
END_GET
END_PROPERTY

{attribute 'monitoring' := 'call'}
PROPERTY Exposure_1us : UDINT
GET
Exposure_1us := THIS^.fbRegExposureTime.Value;
END_GET
SET
IF THIS^.fbRegExposureTime.Value <> Exposure_1us THEN
 	//Set Camera from AQUIRING in OPENED - only on new value
	THIS^.fbCamera.StopAcquisition();
END_IF

THIS^.fbRegExposureTime.Value := Exposure_1us;
END_SET
END_PROPERTY

{attribute 'monitoring' := 'call'}
//IP-Adress as STRING(15)
PROPERTY IPAddress : T_IPv4Addr
GET
VAR
	nValueTemp : UDINT;
	stAdressByteArray   : T_IPv4AddrArr; // Byte-Array
END_VAR

IF SIZEOF(fbRegCurrentIPAddress.Value) <> (4*SIZEOF(BYTE)) THEN
	//Error wrond Datatype, Return 0.0.0.0
	IPAddress := F_CreateIPv4Addr(stAdressByteArray);
	RETURN;
END_IF



//store in a temp variable
nValueTemp := fbRegCurrentIPAddress.Value;


//convert to struct(Array of byte)
Tc2_System.MEMCPY(srcAddr:= ADR(nValueTemp)+3, destAddr:= ADR(stAdressByteArray)+0, n:= SIZEOF(BYTE));
Tc2_System.MEMCPY(srcAddr:= ADR(nValueTemp)+2, destAddr:= ADR(stAdressByteArray)+1, n:= SIZEOF(BYTE));
Tc2_System.MEMCPY(srcAddr:= ADR(nValueTemp)+1, destAddr:= ADR(stAdressByteArray)+2, n:= SIZEOF(BYTE));
Tc2_System.MEMCPY(srcAddr:= ADR(nValueTemp)+0, destAddr:= ADR(stAdressByteArray)+3, n:= SIZEOF(BYTE));


IPAddress := F_CreateIPv4Addr(stAdressByteArray); //Byte-Array to String
END_GET
END_PROPERTY

{attribute 'monitoring' := 'call'}
//MAC-Adress from camera
PROPERTY MacAddress : STRING(12)
GET
IF NOT(fbRegGevMACAddressHighWord.ReadDone AND fbRegGevMACAddressLowWord.ReadDone) THEN
	//Wait for first read
	RETURN;
END_IF

MacAddress := Tc2_Standard.CONCAT(
								//This function converts a decimal number into a hexadecimal string (base 16).
								STR1:= Tc2_Utilities.DWORD_TO_HEXSTR(in:= fbRegGevMACAddressHighWord.Value, iPrecision:= 4, bLoCase:= TRUE ), 
								STR2:= Tc2_Utilities.DWORD_TO_HEXSTR(in:= fbRegGevMACAddressLowWord.Value, iPrecision:= 8, bLoCase:= TRUE )
								);
END_GET
END_PROPERTY

{attribute 'monitoring' := 'call'}
PROPERTY TriggerSource : E_TriggerSource
GET
TriggerSource := THIS^.fbRegTriggerSource.Value;
END_GET
SET
IF THIS^.fbRegTriggerSource.Value <> TriggerSource THEN
 	//Set Camera from AQUIRING in OPENED - only on new value
	THIS^.fbCamera.StopAcquisition();
END_IF

fbRegTriggerSource.Value := TriggerSource;
END_SET
END_PROPERTY

METHOD FB_init : BOOL
VAR_INPUT
	bInitRetains : BOOL; // if TRUE, the retain variables are initialized (warm start / cold start)
	bInCopyCode : BOOL;  // if TRUE, the instance afterwards gets moved into the copy code (online change)
END_VAR
VAR_INST
	{attribute 'hide'}
	bFBInitCalledOnce : BOOL; //Do the following code once during start up and not during onlinechange
END_VAR
//Do the following code once during start up and not during onlinechange
IF NOT bFBInitCalledOnce THEN 
	//Read/Write
	fbVnRegisterList.AddObject(fbRegAcquisitionMode);
	fbVnRegisterList.AddObject(fbRegTriggerMode);
	fbVnRegisterList.AddObject(fbRegTriggerSource);
	fbVnRegisterList.AddObject(fbRegExposureTime);
	fbVnRegisterList.AddObject(fbRegDeviceDefaultState);
	
	//Read only
	fbVnRegisterList.AddObject(fbRegDeviceVendorName);
	fbVnRegisterList.AddObject(fbRegDeviceModelName);
	fbVnRegisterList.AddObject(fbRegDeviceVersion);
	fbVnRegisterList.AddObject(fbRegDeviceSerialNumber);
	fbVnRegisterList.AddObject(fbRegCurrentIPAddress);
	fbVnRegisterList.AddObject(fbRegGevMACAddressHighWord);
	fbVnRegisterList.AddObject(fbRegGevMACAddressLowWord);
	

	
	//Prepare for EtherCat-TimeStamp-Trigger use
	fbRegAcquisitionMode.Value 	:=  16#00; 	//Continous
	fbRegTriggerMode.Value		:=  16#01; 	//ON	 
	fbRegTriggerSource.Value	:=  E_TriggerSource.EtherCAT; 	//EtherCat	 
	fbRegDeviceDefaultState.Value	:=  E_DeviceDefaultState.AutoDetect; 
	fbRegExposureTime.Value	 	:= 	15; 	//[us] smallest allowed value
	
	
END_IF

bFBInitCalledOnce := TRUE;
END_METHOD

//Reference to base function block
PROPERTY GevCameraControl : REFERENCE TO FB_VN_GevCameraControl
GET
GevCameraControl REF= THIS^.fbCamera;
END_GET
END_PROPERTY

METHOD Initialize : HRESULT
VAR 
	fbTaskInfo		 : PlcTaskSystemInfo;
END_VAR
VAR_INST
	//This error cannot be reset. Requires a reset cold
	{attribute 'hide'}	
	fbInitError : FB_TcAlarm;
END_VAR
SUPER^.Initialize();


// Object id of ImagePoovider is not set
IF THIS^.fbCamera.oidITcVnGevImageProvider = 0 THEN
	IF NOT fbInitError.bRaised THEN 
		//This error cannot be reset. Requires a reset cold
		fbInitError.CreateEx(stEventEntry:=TC_EVENTS.CHALET_Vision_Events.ObjectIdNotSet, ipSourceInfo := THIS^.fbSourceInfo, bWithConfirmation := FALSE);
		fbInitError.Raise(0);
	END_IF
	Initialize := E_FAIL;
	RETURN;
END_IF
END_METHOD

{attribute 'monitoring' := 'call'}
PROPERTY OID : CHALET_BaseComponents.OTCID
GET
OID := THIS^.fbCamera.oidITcVnGevImageProvider;
END_GET
END_PROPERTY

METHOD Reset : HRESULT
VAR_INPUT
END_VAR
bResetCommand := TRUE;
END_METHOD

METHOD PUBLIC Softtrigger : HRESULT
(* Check if not in wrong state *)
IF NOT ((THIS^.eState = ETcVnCameraState.TCVN_CS_ACQUIRING) OR (THIS^.eState = ETcVnCameraState.TCVN_CS_OPENED)) THEN
	Softtrigger := E_FAIL;
	RETURN;
END_IF


THIS^.eState := ETcVnCameraState.TCVN_CS_TRIGGERING;

// Trigger image
Softtrigger := fbCamera.TriggerImage();
END_METHOD

{attribute 'monitoring' := 'call'}
PROPERTY State : ETcVnCameraState
GET
State := THIS^.eState;
END_GET
END_PROPERTY

METHOD  TryGetImage : HRESULT
VAR_INPUT
	stImageWithInfo : REFERENCE TO ST_ImageWithInfo;
END_VAR
IF NOT __ISVALIDREF(stImageWithInfo) THEN
	//Error, invalide input
	TryGetImage := E_FAIL;
	RETURN;
END_IF


(* Release the old image before overwriting it with the new one *)	
IF stImageWithInfo.ipImage <> 0 THEN
	FW_SafeRelease(ADR(stImageWithInfo.ipImage));
END_IF

(*  Lock the image to prevent multiple access *)
(*	🔒 LOCKED FROM HERE --------------------------------------------- *)
IF THIS^.fbCrititcalSection.Enter() THEN
	
	(* Get current image from camera *)
	TryGetImage := fbCamera.GetCurrentImageWithGvspInfo(
						ipImage := stImageWithInfo.ipImage,
						stGvspInfo := stImageWithInfo.stGvspInfo
						);

	(* Get image info from received image *)
	F_VN_GetImageInfo(	ipImage:=stImageWithInfo.ipImage, 
						stImageInfo:=stImageWithInfo.stInfo, 
						hrPrev:=TryGetImage );
	
	(* for a camera a fictitious name *)
	stImageWithInfo.sCurrentImageFileName := TO_STRING(stImageWithInfo.stGvspInfo.BlockId);			

	(*	🔓 LOCKED TO HERE ----------------------------------------------- *)
	THIS^.fbCrititcalSection.Leave();
END_IF
END_METHOD

METHOD Update : HRESULT
VAR
	ipVnRegisterStatus : I_VnRegister_Status;
	bAllReadDone : BOOL := TRUE;
	bAllWriteDone : BOOL := TRUE;
END_VAR
(* Get current source state *)					
eState := fbCamera.GetState();

(* Source state machine *)
CASE eState OF
	TCVN_CS_INITIAL, TCVN_CS_INITIALIZING:
		fbFeedback.ActiveCommand := 'InitializeCamera';
		fbFeedback.hr := fbCamera.InitializeCamera();

	TCVN_CS_INITIALIZED,  TCVN_CS_OPENING:
		// Reset all read and write flags 
		THIS^.fbVnRegisterList.ResetIterator();
		WHILE THIS^.fbVnRegisterList.HasNextObject() DO
			//Redo a read oder write for each parameter
			THIS^.fbVnRegisterList.GetNextObject().Initialize();
		END_WHILE
		THIS^.fbVnRegisterList.RestoreIterator();
		
		fbFeedback.ActiveCommand := 'OpenCamera';
		fbFeedback.hr := fbCamera.OpenCamera();
		
	TCVN_CS_OPENED:
		// Read and write all camera parameter in this OPENED-State 
		THIS^.fbVnRegisterList.ResetIterator();
		WHILE THIS^.fbVnRegisterList.HasNextObject() DO
			IF __QUERYINTERFACE(THIS^.fbVnRegisterList.GetNextObject(),ipVnRegisterStatus) THEN
				bAllReadDone := bAllReadDone AND ipVnRegisterStatus.ReadDone;
				bAllWriteDone := bAllWriteDone AND ipVnRegisterStatus.WriteDone;
			END_IF
		END_WHILE
		THIS^.fbVnRegisterList.RestoreIterator();
		
		IF bAllReadDone AND bAllWriteDone THEN
			(* Done - Process with state machine *)
			fbFeedback.ActiveCommand := 'StartAcquisition';
			fbFeedback.hr := fbCamera.StartAcquisition();
		ELSE
			fbFeedback.ActiveCommand := 'ReadWrite Camaera Parameters';
			fbFeedback.Busy	:= TRUE;;
		END_IF
	
		
	TCVN_CS_STARTACQUISITION:
		fbFeedback.ActiveCommand := 'StartAcquisition';
		fbFeedback.hr := fbCamera.StartAcquisition();
		
		
	TCVN_CS_STOPACQUISITION:
		fbFeedback.ActiveCommand := 'StopAcquisition';
		fbFeedback.hr := fbCamera.StopAcquisition();
		
	TCVN_CS_ACQUIRING:
		//wait for trigger
		;
		
	TCVN_CS_TRIGGERING:
		(* Execute the triggering until done *)
		fbFeedback.ActiveCommand := 'TriggerImage';
		fbFeedback.hr := fbCamera.TriggerImage();
		
	TCVN_CS_ERROR:	
	
		(* Reset if commanded *)
		IF THIS^.bResetCommand THEN
			fbFeedback.ActiveCommand := 'Reset';
			fbFeedback.hr := THIS^.fbCamera.Reset();			
		END_IF
END_CASE

(* Clear Alarm if not in Error-State *)
IF eState <> TCVN_CS_ERROR THEN
	THIS^.bResetCommand := FALSE;
END_IF


(* Update camera parameters*)
fbVnRegisterList.Update();
END_METHOD

END_FUNCTION_BLOCK

// COMPONENTs/ImageProvider/Camera/I_GigEVision_Register_Connection
INTERFACE I_GigEVision_Register_Connection

